LIN {X 0,Y 418.253,Z 298.382,A -85,B 0,C 180,E1 -10125.114,E2 -10125.114} C_VEL
LIN {X 0,Y 418.285,Z 298.384,A -85,B 0,C 180,E1 -10127.775,E2 -10127.775} C_VEL
LIN {X 0,Y 418.259,Z 298.386,A -85,B 0,C 180,E1 -10131.561,E2 -10131.561} C_VEL
LIN {X 0,Y 418.254,Z 298.387,A -85,B 0,C 180,E1 -10135.161,E2 -10135.161} C_VEL
LIN {X 0,Y 418.24,Z 298.388,A -85,B 0,C 180,E1 -10137.474,E2 -10137.474} C_VEL
LIN {X 0,Y 418.265,Z 298.384,A -85,B 0,C 180,E1 -10140.897,E2 -10140.897} C_VEL
LIN {X 0,Y 418.312,Z 298.534,A -85,B 0,C 180,E1 -10141.838,E2 -10141.838} C_VEL
LIN {X 0,Y 420.829,Z 310.049,A -85,B 0,C 180,E1 -10144.399,E2 -10144.399} C_VEL
LIN {X 0,Y 421.677,Z 315.896,A -85,B 0,C 180,E1 -10145.64,E2 -10145.64} C_VEL
LIN {X 0,Y 420.473,Z 332.793,A -85,B 0,C 180,E1 -10148.941,E2 -10148.941} C_VEL
LIN {X 0,Y 419.947,Z 341.283,A -85,B 0,C 180,E1 -10150.58,E2 -10150.58} C_VEL
LIN {X 0,Y 423.915,Z 364.649,A -85,B 0,C 180,E1 -10151.228,E2 -10151.228} C_VEL
LIN {X 0,Y 424.429,Z 370.899,A -85,B 0,C 180,E1 -10151.367,E2 -10151.367} C_VEL
LIN {X 0,Y 423.375,Z 450.721,A -85,B 0,C 180,E1 -10152.772,E2 -10152.772} C_VEL
LIN {X 0,Y 422.75,Z 464.397,A -85,B 0,C 180,E1 -10153.213,E2 -10153.213} C_VEL
LIN {X 0,Y 422.113,Z 476.708,A -85,B 0,C 180,E1 -10153.808,E2 -10153.808} C_VEL
LIN {X 0,Y 421.326,Z 487.75,A -85,B 0,C 180,E1 -10154.522,E2 -10154.522} C_VEL
LIN {X 0,Y 420.546,Z 499.288,A -85,B 0,C 180,E1 -10155.484,E2 -10155.484} C_VEL
LIN {X 0,Y 419.713,Z 509.697,A -85,B 0,C 180,E1 -10156.567,E2 -10156.567} C_VEL
LIN {X 0,Y 419.106,Z 518.223,A -85,B 0,C 180,E1 -10157.656,E2 -10157.656} C_VEL
LIN {X 0,Y 418.404,Z 526.105,A -85,B 0,C 180,E1 -10158.864,E2 -10158.864} C_VEL
LIN {X 0,Y 417.832,Z 533.825,A -85,B 0,C 180,E1 -10160.318,E2 -10160.318} C_VEL
LIN {X 0,Y 417.461,Z 540.039,A -85,B 0,C 180,E1 -10161.774,E2 -10161.774} C_VEL
LIN {X 0,Y 417.233,Z 544.991,A -85,B 0,C 180,E1 -10163.23,E2 -10163.23} C_VEL
LIN {X 0,Y 417.12,Z 548.824,A -85,B 0,C 180,E1 -10164.684,E2 -10164.684} C_VEL
LIN {X 0,Y 417.015,Z 551.638,A -85,B 0,C 180,E1 -10166.136,E2 -10166.136} C_VEL
LIN {X 0,Y 417.069,Z 553.918,A -85,B 0,C 180,E1 -10168.07,E2 -10168.07} C_VEL
LIN {X 0,Y 417.013,Z 554.462,A -85,B 0,C 180,E1 -10169.036,E2 -10169.036} C_VEL
LIN {X 0,Y 417.027,Z 554.574,A -85,B 0,C 180,E1 -10170.001,E2 -10170.001} C_VEL
LIN {X 0,Y 417.073,Z 553.627,A -85,B 0,C 180,E1 -10171.933,E2 -10171.933} C_VEL
LIN {X 0,Y 417.061,Z 552.561,A -85,B 0,C 180,E1 -10172.899,E2 -10172.899} C_VEL
LIN {X 0,Y 417.018,Z 551.035,A -85,B 0,C 180,E1 -10173.867,E2 -10173.867} C_VEL
LIN {X 0,Y 417.122,Z 547.958,A -85,B 0,C 180,E1 -10175.319,E2 -10175.319} C_VEL
LIN {X 0,Y 417.233,Z 543.806,A -85,B 0,C 180,E1 -10176.773,E2 -10176.773} C_VEL
LIN {X 0,Y 417.496,Z 537.449,A -85,B 0,C 180,E1 -10178.472,E2 -10178.472} C_VEL
LIN {X 0,Y 417.865,Z 530.518,A -85,B 0,C 180,E1 -10179.928,E2 -10179.928} C_VEL
LIN {X 0,Y 418.277,Z 523.434,A -85,B 0,C 180,E1 -10181.142,E2 -10181.142} C_VEL
LIN {X 0,Y 418.885,Z 514.891,A -85,B 0,C 180,E1 -10182.353,E2 -10182.353} C_VEL
LIN {X 0,Y 419.584,Z 504.318,A -85,B 0,C 180,E1 -10183.563,E2 -10183.563} C_VEL
LIN {X 0,Y 420.222,Z 492.389,A -85,B 0,C 180,E1 -10184.654,E2 -10184.654} C_VEL
LIN {X 0,Y 420.969,Z 480.36,A -85,B 0,C 180,E1 -10185.494,E2 -10185.494} C_VEL
LIN {X 0,Y 421.575,Z 467.817,A -85,B 0,C 180,E1 -10186.154,E2 -10186.154} C_VEL
LIN {X 0,Y 422.144,Z 454.764,A -85,B 0,C 180,E1 -10186.628,E2 -10186.628} C_VEL
LIN {X 0,Y 422.485,Z 438.987,A -85,B 0,C 180,E1 -10186.957,E2 -10186.957} C_VEL
LIN {X 0,Y 423.146,Z 367.635,A -85,B 0,C 180,E1 -10188.174,E2 -10188.174} C_VEL
LIN {X 0,Y 419.379,Z 341.81,A -85,B 0,C 180,E1 -10188.774,E2 -10188.774} C_VEL
LIN {X 0,Y 420.377,Z 324.387,A -85,B 0,C 180,E1 -10192.097,E2 -10192.097} C_VEL
LIN {X 0,Y 421.059,Z 313.774,A -85,B 0,C 180,E1 -10194.139,E2 -10194.139} C_VEL
LIN {X 0,Y 420.155,Z 307.557,A -85,B 0,C 180,E1 -10195.408,E2 -10195.408} C_VEL
LIN {X 0,Y 418.343,Z 298.376,A -85,B 0,C 180,E1 -10197.364,E2 -10197.364} C_VEL
LIN {X 0,Y 418.245,Z 298.384,A -85,B 0,C 180,E1 -10201.02,E2 -10201.02} C_VEL
LIN {X 0,Y 418.253,Z 298.382,A -85,B 0,C 180,E1 -10203.678,E2 -10203.678} C_VEL
LIN {X 0,Y 418.245,Z 298.382,A -85,B 0,C 180,E1 -10207.225,E2 -10207.225} C_VEL
LIN {X 0,Y 418.249,Z 298.382,A -85,B 0,C 180,E1 -10209.683,E2 -10209.683} C_VEL
LIN {X 0,Y 418.235,Z 298.388,A -85,B 0,C 180,E1 -10212.322,E2 -10212.322} C_VEL
LIN {X 0,Y 418.242,Z 298.384,A -85,B 0,C 180,E1 -10215.109,E2 -10215.109} C_VEL
LIN {X 0,Y 418.246,Z 298.382,A -85,B 0,C 180,E1 -10217.767,E2 -10217.767} C_VEL
LIN {X 0,Y 418.255,Z 298.386,A -85,B 0,C 180,E1 -10220.62,E2 -10220.62} C_VEL
LIN {X 0,Y 418.248,Z 298.381,A -85,B 0,C 180,E1 -10223.976,E2 -10223.976} C_VEL
LIN {X 0,Y 418.249,Z 298.384,A -85,B 0,C 180,E1 -10227.472,E2 -10227.472} C_VEL
LIN {X 0,Y 418.275,Z 298.383,A -85,B 0,C 180,E1 -10230.896,E2 -10230.896} C_VEL
LIN {X 0,Y 418.275,Z 298.378,A -85,B 0,C 180,E1 -10234.096,E2 -10234.096} C_VEL
LIN {X 0,Y 418.238,Z 298.389,A -85,B 0,C 180,E1 -10237.264,E2 -10237.264} C_VEL
LIN {X 0,Y 418.289,Z 298.376,A -85,B 0,C 180,E1 -10240.364,E2 -10240.364} C_VEL
LIN {X 0,Y 418.323,Z 298.378,A -85,B 0,C 180,E1 -10243.405,E2 -10243.405} C_VEL
LIN {X 0,Y 418.353,Z 298.369,A -85,B 0,C 180,E1 -10246.999,E2 -10246.999} C_VEL
LIN {X 0,Y 418.345,Z 298.371,A -85,B 0,C 180,E1 -10250.329,E2 -10250.329} C_VEL
LIN {X 0,Y 418.452,Z 298.357,A -85,B 0,C 180,E1 -10253.248,E2 -10253.248} C_VEL
LIN {X 0,Y 418.339,Z 298.37,A -85,B 0,C 180,E1 -10255.181,E2 -10255.181} C_VEL
LIN {X 0,Y 418.548,Z 298.352,A -85,B 0,C 180,E1 -10258.075,E2 -10258.075} C_VEL
LIN {X 0,Y 418.674,Z 298.335,A -85,B 0,C 180,E1 -10260,E2 -10260} C_VEL
LIN {X 0,Y 418.504,Z 298.35,A -85,B 0,C 180,E1 -10262.888,E2 -10262.888} C_VEL
LIN {X 0,Y 418.474,Z 298.355,A -85,B 0,C 180,E1 -10266.629,E2 -10266.629} C_VEL
LIN {X 0,Y 418.344,Z 298.37,A -85,B 0,C 180,E1 -10269.671,E2 -10269.671} C_VEL
LIN {X 0,Y 418.352,Z 298.371,A -85,B 0,C 180,E1 -10273,E2 -10273} C_VEL
LIN {X 0,Y 418.318,Z 298.38,A -85,B 0,C 180,E1 -10276.735,E2 -10276.735} C_VEL
LIN {X 0,Y 418.276,Z 298.378,A -85,B 0,C 180,E1 -10279.789,E2 -10279.789} C_VEL
LIN {X 0,Y 418.237,Z 298.389,A -85,B 0,C 180,E1 -10282.736,E2 -10282.736} C_VEL
LIN {X 0,Y 418.276,Z 298.378,A -85,B 0,C 180,E1 -10285.904,E2 -10285.904} C_VEL
LIN {X 0,Y 418.27,Z 298.385,A -85,B 0,C 180,E1 -10289.161,E2 -10289.161} C_VEL
LIN {X 0,Y 418.262,Z 298.383,A -85,B 0,C 180,E1 -10292.843,E2 -10292.843} C_VEL
LIN {X 0,Y 418.248,Z 298.381,A -85,B 0,C 180,E1 -10296.237,E2 -10296.237} C_VEL
LIN {X 0,Y 418.255,Z 298.385,A -85,B 0,C 180,E1 -10299.681,E2 -10299.681} C_VEL
LIN {X 0,Y 418.234,Z 298.383,A -85,B 0,C 180,E1 -10302.32,E2 -10302.32} C_VEL
LIN {X 0,Y 418.24,Z 298.385,A -85,B 0,C 180,E1 -10305.108,E2 -10305.108} C_VEL
LIN {X 0,Y 418.243,Z 298.389,A -85,B 0,C 180,E1 -10307.766,E2 -10307.766} C_VEL
LIN {X 0,Y 418.249,Z 298.381,A -85,B 0,C 180,E1 -10310.62,E2 -10310.62} C_VEL
LIN {X 0,Y 418.247,Z 298.388,A -85,B 0,C 180,E1 -10313.975,E2 -10313.975} C_VEL
LIN {X 0,Y 418.261,Z 298.38,A -85,B 0,C 180,E1 -10317.155,E2 -10317.155} C_VEL
LIN {X 0,Y 418.272,Z 298.379,A -85,B 0,C 180,E1 -10320.894,E2 -10320.894} C_VEL
LIN {X 0,Y 418.272,Z 298.385,A -85,B 0,C 180,E1 -10324.095,E2 -10324.095} C_VEL
LIN {X 0,Y 418.241,Z 298.382,A -85,B 0,C 180,E1 -10327.263,E2 -10327.263} C_VEL
LIN {X 0,Y 418.319,Z 298.38,A -85,B 0,C 180,E1 -10330.365,E2 -10330.365} C_VEL
LIN {X 0,Y 418.32,Z 298.372,A -85,B 0,C 180,E1 -10333.403,E2 -10333.403} C_VEL
LIN {X 0,Y 418.348,Z 298.372,A -85,B 0,C 180,E1 -10336.998,E2 -10336.998} C_VEL
LIN {X 0,Y 418.34,Z 298.373,A -85,B 0,C 180,E1 -10340.327,E2 -10340.327} C_VEL
LIN {X 0,Y 418.457,Z 298.388,A -85,B 0,C 180,E1 -10343.121,E2 -10343.121} C_VEL
LIN {X 0,Y 419.862,Z 307.44,A -85,B 0,C 180,E1 -10345.198,E2 -10345.198} C_VEL
LIN {X 0,Y 419.717,Z 312.544,A -85,B 0,C 180,E1 -10346.308,E2 -10346.308} C_VEL
LIN {X 0,Y 423.532,Z 333.046,A -85,B 0,C 180,E1 -10346.824,E2 -10346.824} C_VEL
LIN {X 0,Y 422.396,Z 420.515,A -85,B 0,C 180,E1 -10348.335,E2 -10348.335} C_VEL
LIN {X 0,Y 422.141,Z 430.007,A -85,B 0,C 180,E1 -10348.618,E2 -10348.618} C_VEL
LIN {X 0,Y 421.418,Z 435.689,A -85,B 0,C 180,E1 -10348.815,E2 -10348.815} C_VEL
LIN {X 0,Y 418.342,Z 444.777,A -85,B 0,C 180,E1 -10349.157,E2 -10349.157} C_VEL
LIN {X 0,Y 415.083,Z 453.573,A -85,B 0,C 180,E1 -10349.603,E2 -10349.603} C_VEL
LIN {X 0,Y 414.083,Z 458.797,A -85,B 0,C 180,E1 -10349.96,E2 -10349.96} C_VEL
LIN {X 0,Y 413.337,Z 470.545,A -85,B 0,C 180,E1 -10350.973,E2 -10350.973} C_VEL
LIN {X 0,Y 412.59,Z 480.693,A -85,B 0,C 180,E1 -10352.073,E2 -10352.073} C_VEL
LIN {X 0,Y 411.883,Z 490.629,A -85,B 0,C 180,E1 -10353.422,E2 -10353.422} C_VEL
LIN {X 0,Y 411.278,Z 499.38,A -85,B 0,C 180,E1 -10354.9,E2 -10354.9} C_VEL
LIN {X 0,Y 410.901,Z 506.355,A -85,B 0,C 180,E1 -10356.382,E2 -10356.382} C_VEL
LIN {X 0,Y 410.522,Z 511.96,A -85,B 0,C 180,E1 -10357.87,E2 -10357.87} C_VEL
LIN {X 0,Y 410.249,Z 516.367,A -85,B 0,C 180,E1 -10359.365,E2 -10359.365} C_VEL
LIN {X 0,Y 410.086,Z 519.69,A -85,B 0,C 180,E1 -10360.865,E2 -10360.865} C_VEL
LIN {X 0,Y 409.94,Z 521.881,A -85,B 0,C 180,E1 -10362.258,E2 -10362.258} C_VEL
LIN {X 0,Y 409.84,Z 523.379,A -85,B 0,C 180,E1 -10363.889,E2 -10363.889} C_VEL
LIN {X 0,Y 409.853,Z 523.751,A -85,B 0,C 180,E1 -10364.903,E2 -10364.903} C_VEL
LIN {X 0,Y 409.855,Z 523.645,A -85,B 0,C 180,E1 -10366.207,E2 -10366.207} C_VEL
LIN {X 0,Y 409.93,Z 522.359,A -85,B 0,C 180,E1 -10367.973,E2 -10367.973} C_VEL
LIN {X 0,Y 410.158,Z 520.14,A -85,B 0,C 180,E1 -10369.539,E2 -10369.539} C_VEL
LIN {X 0,Y 410.355,Z 516.918,A -85,B 0,C 180,E1 -10371.077,E2 -10371.077} C_VEL
LIN {X 0,Y 410.73,Z 512.238,A -85,B 0,C 180,E1 -10372.716,E2 -10372.716} C_VEL
LIN {X 0,Y 411.197,Z 506.699,A -85,B 0,C 180,E1 -10374.215,E2 -10374.215} C_VEL
LIN {X 0,Y 411.84,Z 499.345,A -85,B 0,C 180,E1 -10375.793,E2 -10375.793} C_VEL
LIN {X 0,Y 412.55,Z 491.704,A -85,B 0,C 180,E1 -10377.108,E2 -10377.108} C_VEL
LIN {X 0,Y 413.388,Z 482.313,A -85,B 0,C 180,E1 -10378.424,E2 -10378.424} C_VEL
LIN {X 0,Y 414.076,Z 473.077,A -85,B 0,C 180,E1 -10379.484,E2 -10379.484} C_VEL
LIN {X 0,Y 414.997,Z 461.664,A -85,B 0,C 180,E1 -10380.532,E2 -10380.532} C_VEL
LIN {X 0,Y 415.769,Z 449.638,A -85,B 0,C 180,E1 -10381.387,E2 -10381.387} C_VEL
LIN {X 0,Y 416.379,Z 437.805,A -85,B 0,C 180,E1 -10382.022,E2 -10382.022} C_VEL
LIN {X 0,Y 416.819,Z 425.374,A -85,B 0,C 180,E1 -10382.496,E2 -10382.496} C_VEL
LIN {X 0,Y 417.163,Z 410.81,A -85,B 0,C 180,E1 -10382.818,E2 -10382.818} C_VEL
LIN {X 0,Y 418.122,Z 333.025,A -85,B 0,C 180,E1 -10384.188,E2 -10384.188} C_VEL
LIN {X 0,Y 414.056,Z 315.081,A -85,B 0,C 180,E1 -10384.753,E2 -10384.753} C_VEL
LIN {X 0,Y 413.542,Z 312.748,A -85,B 0,C 180,E1 -10384.864,E2 -10384.864} C_VEL
LIN {X 0,Y 413.307,Z 309.399,A -85,B 0,C 180,E1 -10385.616,E2 -10385.616} C_VEL
LIN {X 0,Y 411.168,Z 299.271,A -85,B 0,C 180,E1 -10388.079,E2 -10388.079} C_VEL
LIN {X 0,Y 411.136,Z 299.271,A -85,B 0,C 180,E1 -10391.224,E2 -10391.224} C_VEL
LIN {X 0,Y 411.163,Z 299.268,A -85,B 0,C 180,E1 -10394.489,E2 -10394.489} C_VEL
LIN {X 0,Y 411.151,Z 299.269,A -85,B 0,C 180,E1 -10398.192,E2 -10398.192} C_VEL
LIN {X 0,Y 411.178,Z 299.27,A -85,B 0,C 180,E1 -10401.833,E2 -10401.833} C_VEL
LIN {X 0,Y 411.195,Z 299.251,A -85,B 0,C 180,E1 -10405.121,E2 -10405.121} C_VEL
LIN {X 0,Y 411.152,Z 299.268,A -85,B 0,C 180,E1 -10408.002,E2 -10408.002} C_VEL
LIN {X 0,Y 411.181,Z 299.266,A -85,B 0,C 180,E1 -10411.407,E2 -10411.407} C_VEL
LIN {X 0,Y 411.213,Z 299.256,A -85,B 0,C 180,E1 -10414.929,E2 -10414.929} C_VEL
LIN {X 0,Y 411.19,Z 299.266,A -85,B 0,C 180,E1 -10417.913,E2 -10417.913} C_VEL
LIN {X 0,Y 411.207,Z 299.26,A -85,B 0,C 180,E1 -10421.051,E2 -10421.051} C_VEL
LIN {X 0,Y 411.239,Z 299.256,A -85,B 0,C 180,E1 -10424.131,E2 -10424.131} C_VEL
LIN {X 0,Y 411.288,Z 299.246,A -85,B 0,C 180,E1 -10427.165,E2 -10427.165} C_VEL
LIN {X 0,Y 411.289,Z 299.254,A -85,B 0,C 180,E1 -10430.161,E2 -10430.161} C_VEL
LIN {X 0,Y 411.408,Z 299.228,A -85,B 0,C 180,E1 -10433.132,E2 -10433.132} C_VEL
LIN {X 0,Y 411.291,Z 299.25,A -85,B 0,C 180,E1 -10435.099,E2 -10435.099} C_VEL
LIN {X 0,Y 411.497,Z 299.22,A -85,B 0,C 180,E1 -10438.043,E2 -10438.043} C_VEL
LIN {X 0,Y 411.626,Z 299.206,A -85,B 0,C 180,E1 -10440,E2 -10440} C_VEL
LIN {X 0,Y 411.443,Z 299.224,A -85,B 0,C 180,E1 -10442.938,E2 -10442.938} C_VEL
LIN {X 0,Y 411.444,Z 299.23,A -85,B 0,C 180,E1 -10446.867,E2 -10446.867} C_VEL
LIN {X 0,Y 411.341,Z 299.24,A -85,B 0,C 180,E1 -10448.846,E2 -10448.846} C_VEL
LIN {X 0,Y 411.271,Z 299.251,A -85,B 0,C 180,E1 -10451.833,E2 -10451.833} C_VEL
LIN {X 0,Y 411.246,Z 299.254,A -85,B 0,C 180,E1 -10454.853,E2 -10454.853} C_VEL
LIN {X 0,Y 411.239,Z 299.252,A -85,B 0,C 180,E1 -10457.916,E2 -10457.916} C_VEL
LIN {X 0,Y 411.183,Z 299.269,A -85,B 0,C 180,E1 -10461.035,E2 -10461.035} C_VEL
LIN {X 0,Y 411.214,Z 299.254,A -85,B 0,C 180,E1 -10464.216,E2 -10464.216} C_VEL
LIN {X 0,Y 411.248,Z 299.252,A -85,B 0,C 180,E1 -10467.479,E2 -10467.479} C_VEL
LIN {X 0,Y 411.191,Z 299.266,A -85,B 0,C 180,E1 -10470.848,E2 -10470.848} C_VEL
LIN {X 0,Y 411.196,Z 299.263,A -85,B 0,C 180,E1 -10474.335,E2 -10474.335} C_VEL
LIN {X 0,Y 411.195,Z 299.264,A -85,B 0,C 180,E1 -10477.974,E2 -10477.974} C_VEL
LIN {X 0,Y 411.192,Z 299.269,A -85,B 0,C 180,E1 -10481.236,E2 -10481.236} C_VEL
LIN {X 0,Y 411.18,Z 299.262,A -85,B 0,C 180,E1 -10484.49,E2 -10484.49} C_VEL
LIN {X 0,Y 411.222,Z 299.257,A -85,B 0,C 180,E1 -10487.299,E2 -10487.299} C_VEL
LIN {X 0,Y 411.224,Z 299.257,A -85,B 0,C 180,E1 -10490.779,E2 -10490.779} C_VEL
LIN {X 0,Y 411.194,Z 299.266,A -85,B 0,C 180,E1 -10494.473,E2 -10494.473} C_VEL
LIN {X 0,Y 411.202,Z 299.262,A -85,B 0,C 180,E1 -10496.875,E2 -10496.875} C_VEL
LIN {X 0,Y 411.229,Z 299.259,A -85,B 0,C 180,E1 -10500.646,E2 -10500.646} C_VEL
LIN {X 0,Y 411.294,Z 299.423,A -85,B 0,C 180,E1 -10501.494,E2 -10501.494} C_VEL
LIN {X 0,Y 413.863,Z 311.135,A -85,B 0,C 180,E1 -10504.161,E2 -10504.161} C_VEL
LIN {X 0,Y 414.801,Z 317.201,A -85,B 0,C 180,E1 -10505.476,E2 -10505.476} C_VEL
LIN {X 0,Y 413.55,Z 334.086,A -85,B 0,C 180,E1 -10508.832,E2 -10508.832} C_VEL
LIN {X 0,Y 413.076,Z 341.056,A -85,B 0,C 180,E1 -10510.203,E2 -10510.203} C_VEL
LIN {X 0,Y 417.161,Z 364.626,A -85,B 0,C 180,E1 -10510.867,E2 -10510.867} C_VEL
LIN {X 0,Y 417.815,Z 370.654,A -85,B 0,C 180,E1 -10511.013,E2 -10511.013} C_VEL
LIN {X 0,Y 416.687,Z 449.899,A -85,B 0,C 180,E1 -10512.423,E2 -10512.423} C_VEL
LIN {X 0,Y 416.097,Z 463.747,A -85,B 0,C 180,E1 -10512.873,E2 -10512.873} C_VEL
LIN {X 0,Y 415.395,Z 476.174,A -85,B 0,C 180,E1 -10513.476,E2 -10513.476} C_VEL
LIN {X 0,Y 414.513,Z 488.07,A -85,B 0,C 180,E1 -10514.261,E2 -10514.261} C_VEL
LIN {X 0,Y 413.672,Z 499.486,A -85,B 0,C 180,E1 -10515.238,E2 -10515.238} C_VEL
LIN {X 0,Y 412.786,Z 509.803,A -85,B 0,C 180,E1 -10516.337,E2 -10516.337} C_VEL
LIN {X 0,Y 412.147,Z 518.256,A -85,B 0,C 180,E1 -10517.444,E2 -10517.444} C_VEL
LIN {X 0,Y 411.295,Z 527.442,A -85,B 0,C 180,E1 -10518.918,E2 -10518.918} C_VEL
LIN {X 0,Y 410.739,Z 534.855,A -85,B 0,C 180,E1 -10520.398,E2 -10520.398} C_VEL
LIN {X 0,Y 410.321,Z 541.71,A -85,B 0,C 180,E1 -10522.126,E2 -10522.126} C_VEL
LIN {X 0,Y 410.042,Z 546.679,A -85,B 0,C 180,E1 -10523.777,E2 -10523.777} C_VEL
LIN {X 0,Y 410.018,Z 549.704,A -85,B 0,C 180,E1 -10525.085,E2 -10525.085} C_VEL
LIN {X 0,Y 409.928,Z 552.753,A -85,B 0,C 180,E1 -10527.053,E2 -10527.053} C_VEL
LIN {X 0,Y 409.996,Z 553.685,A -85,B 0,C 180,E1 -10528.037,E2 -10528.037} C_VEL
LIN {X 0,Y 409.938,Z 554.208,A -85,B 0,C 180,E1 -10529.019,E2 -10529.019} C_VEL
LIN {X 0,Y 409.948,Z 554.302,A -85,B 0,C 180,E1 -10530.001,E2 -10530.001} C_VEL
LIN {X 0,Y 410.001,Z 553.331,A -85,B 0,C 180,E1 -10531.966,E2 -10531.966} C_VEL
LIN {X 0,Y 409.959,Z 552.242,A -85,B 0,C 180,E1 -10532.949,E2 -10532.949} C_VEL
LIN {X 0,Y 409.937,Z 550.698,A -85,B 0,C 180,E1 -10533.934,E2 -10533.934} C_VEL
LIN {X 0,Y 410.019,Z 547.59,A -85,B 0,C 180,E1 -10535.411,E2 -10535.411} C_VEL
LIN {X 0,Y 410.165,Z 543.409,A -85,B 0,C 180,E1 -10536.89,E2 -10536.89} C_VEL
LIN {X 0,Y 410.426,Z 537.017,A -85,B 0,C 180,E1 -10538.619,E2 -10538.619} C_VEL
LIN {X 0,Y 410.806,Z 530.047,A -85,B 0,C 180,E1 -10540.101,E2 -10540.101} C_VEL
LIN {X 0,Y 411.379,Z 521.302,A -85,B 0,C 180,E1 -10541.581,E2 -10541.581} C_VEL
LIN {X 0,Y 412.001,Z 512.334,A -85,B 0,C 180,E1 -10542.814,E2 -10542.814} C_VEL
LIN {X 0,Y 412.653,Z 502.834,A -85,B 0,C 180,E1 -10543.883,E2 -10543.883} C_VEL
LIN {X 0,Y 413.329,Z 491.621,A -85,B 0,C 180,E1 -10544.904,E2 -10544.904} C_VEL
LIN {X 0,Y 414.103,Z 479.435,A -85,B 0,C 180,E1 -10545.758,E2 -10545.758} C_VEL
LIN {X 0,Y 414.764,Z 466.689,A -85,B 0,C 180,E1 -10546.426,E2 -10546.426} C_VEL
LIN {X 0,Y 415.272,Z 454.102,A -85,B 0,C 180,E1 -10546.88,E2 -10546.88} C_VEL
LIN {X 0,Y 415.595,Z 438.077,A -85,B 0,C 180,E1 -10547.215,E2 -10547.215} C_VEL
LIN {X 0,Y 416.208,Z 367.341,A -85,B 0,C 180,E1 -10548.443,E2 -10548.443} C_VEL
LIN {X 0,Y 412.425,Z 341.549,A -85,B 0,C 180,E1 -10549.054,E2 -10549.054} C_VEL
LIN {X 0,Y 413.409,Z 325.2,A -85,B 0,C 180,E1 -10552.227,E2 -10552.227} C_VEL
LIN {X 0,Y 414.081,Z 314.581,A -85,B 0,C 180,E1 -10554.306,E2 -10554.306} C_VEL
LIN {X 0,Y 412.855,Z 307.049,A -85,B 0,C 180,E1 -10555.878,E2 -10555.878} C_VEL
LIN {X 0,Y 411.318,Z 299.252,A -85,B 0,C 180,E1 -10557.578,E2 -10557.578} C_VEL
LIN {X 0,Y 411.188,Z 299.262,A -85,B 0,C 180,E1 -10561.284,E2 -10561.284} C_VEL
LIN {X 0,Y 411.211,Z 299.265,A -85,B 0,C 180,E1 -10564.334,E2 -10564.334} C_VEL
LIN {X 0,Y 411.196,Z 299.263,A -85,B 0,C 180,E1 -10567.975,E2 -10567.975} C_VEL
LIN {X 0,Y 411.169,Z 299.264,A -85,B 0,C 180,E1 -10571.229,E2 -10571.229} C_VEL
LIN {X 0,Y 411.182,Z 299.268,A -85,B 0,C 180,E1 -10574.491,E2 -10574.491} C_VEL
LIN {X 0,Y 411.183,Z 299.263,A -85,B 0,C 180,E1 -10578.195,E2 -10578.195} C_VEL
LIN {X 0,Y 411.22,Z 299.264,A -85,B 0,C 180,E1 -10580.776,E2 -10580.776} C_VEL
LIN {X 0,Y 411.201,Z 299.262,A -85,B 0,C 180,E1 -10584.471,E2 -10584.471} C_VEL
LIN {X 0,Y 411.211,Z 299.264,A -85,B 0,C 180,E1 -10586.874,E2 -10586.874} C_VEL
LIN {X 0,Y 411.239,Z 299.256,A -85,B 0,C 180,E1 -10590.644,E2 -10590.644} C_VEL
LIN {X 0,Y 411.244,Z 299.257,A -85,B 0,C 180,E1 -10593.619,E2 -10593.619} C_VEL
LIN {X 0,Y 411.203,Z 299.261,A -85,B 0,C 180,E1 -10596.852,E2 -10596.852} C_VEL
LIN {X 0,Y 411.221,Z 299.258,A -85,B 0,C 180,E1 -10600.051,E2 -10600.051} C_VEL
LIN {X 0,Y 411.27,Z 299.253,A -85,B 0,C 180,E1 -10603.131,E2 -10603.131} C_VEL
LIN {X 0,Y 411.312,Z 299.246,A -85,B 0,C 180,E1 -10606.896,E2 -10606.896} C_VEL
LIN {X 0,Y 411.297,Z 299.25,A -85,B 0,C 180,E1 -10610.161,E2 -10610.161} C_VEL
LIN {X 0,Y 411.401,Z 299.235,A -85,B 0,C 180,E1 -10613.132,E2 -10613.132} C_VEL
LIN {X 0,Y 411.309,Z 299.246,A -85,B 0,C 180,E1 -10615.099,E2 -10615.099} C_VEL
LIN {X 0,Y 411.517,Z 299.228,A -85,B 0,C 180,E1 -10618.042,E2 -10618.042} C_VEL
LIN {X 0,Y 411.643,Z 299.211,A -85,B 0,C 180,E1 -10620,E2 -10620} C_VEL
LIN {X 0,Y 411.461,Z 299.227,A -85,B 0,C 180,E1 -10622.937,E2 -10622.937} C_VEL
LIN {X 0,Y 411.437,Z 299.23,A -85,B 0,C 180,E1 -10626.629,E2 -10626.629} C_VEL
LIN {X 0,Y 411.324,Z 299.246,A -85,B 0,C 180,E1 -10628.846,E2 -10628.846} C_VEL
LIN {X 0,Y 411.288,Z 299.249,A -85,B 0,C 180,E1 -10631.832,E2 -10631.832} C_VEL
LIN {X 0,Y 411.266,Z 299.256,A -85,B 0,C 180,E1 -10634.852,E2 -10634.852} C_VEL
LIN {X 0,Y 411.251,Z 299.253,A -85,B 0,C 180,E1 -10637.915,E2 -10637.915} C_VEL
LIN {X 0,Y 411.201,Z 299.264,A -85,B 0,C 180,E1 -10641.034,E2 -10641.034} C_VEL
LIN {X 0,Y 411.226,Z 299.257,A -85,B 0,C 180,E1 -10644.215,E2 -10644.215} C_VEL
LIN {X 0,Y 411.264,Z 299.254,A -85,B 0,C 180,E1 -10647.477,E2 -10647.477} C_VEL
LIN {X 0,Y 411.194,Z 299.264,A -85,B 0,C 180,E1 -10650.847,E2 -10650.847} C_VEL
LIN {X 0,Y 411.21,Z 299.258,A -85,B 0,C 180,E1 -10654.333,E2 -10654.333} C_VEL
LIN {X 0,Y 411.199,Z 299.261,A -85,B 0,C 180,E1 -10657.973,E2 -10657.973} C_VEL
LIN {X 0,Y 411.186,Z 299.261,A -85,B 0,C 180,E1 -10660.503,E2 -10660.503} C_VEL
LIN {X 0,Y 411.178,Z 299.265,A -85,B 0,C 180,E1 -10663.133,E2 -10663.133} C_VEL
LIN {X 0,Y 411.172,Z 299.267,A -85,B 0,C 180,E1 -10665.88,E2 -10665.88} C_VEL
LIN {X 0,Y 411.167,Z 299.263,A -85,B 0,C 180,E1 -10668.771,E2 -10668.771} C_VEL
LIN {X 0,Y 411.195,Z 299.265,A -85,B 0,C 180,E1 -10672.025,E2 -10672.025} C_VEL
LIN {X 0,Y 411.21,Z 299.263,A -85,B 0,C 180,E1 -10675.666,E2 -10675.666} C_VEL
LIN {X 0,Y 411.193,Z 299.26,A -85,B 0,C 180,E1 -10679.151,E2 -10679.151} C_VEL
LIN {X 0,Y 411.262,Z 299.255,A -85,B 0,C 180,E1 -10682.521,E2 -10682.521} C_VEL
LIN {X 0,Y 411.229,Z 299.258,A -85,B 0,C 180,E1 -10685.783,E2 -10685.783} C_VEL
LIN {X 0,Y 411.205,Z 299.26,A -85,B 0,C 180,E1 -10688.965,E2 -10688.965} C_VEL
LIN {X 0,Y 411.255,Z 299.255,A -85,B 0,C 180,E1 -10692.084,E2 -10692.084} C_VEL
LIN {X 0,Y 411.262,Z 299.253,A -85,B 0,C 180,E1 -10695.146,E2 -10695.146} C_VEL
LIN {X 0,Y 411.286,Z 299.251,A -85,B 0,C 180,E1 -10698.166,E2 -10698.166} C_VEL
LIN {X 0,Y 411.438,Z 299.236,A -85,B 0,C 180,E1 -10702.191,E2 -10702.191} C_VEL
LIN {X 0,Y 411.4,Z 299.304,A -85,B 0,C 180,E1 -10702.941,E2 -10702.941} C_VEL
LIN {X 0,Y 412.773,Z 307.583,A -85,B 0,C 180,E1 -10704.87,E2 -10704.87} C_VEL
LIN {X 0,Y 412.749,Z 312.82,A -85,B 0,C 180,E1 -10706.032,E2 -10706.032} C_VEL
LIN {X 0,Y 416.688,Z 333.567,A -85,B 0,C 180,E1 -10706.566,E2 -10706.566} C_VEL
LIN {X 0,Y 415.539,Z 420.703,A -85,B 0,C 180,E1 -10708.094,E2 -10708.094} C_VEL
LIN {X 0,Y 415.127,Z 434.046,A -85,B 0,C 180,E1 -10708.532,E2 -10708.532} C_VEL
LIN {X 0,Y 414.743,Z 446.232,A -85,B 0,C 180,E1 -10709.126,E2 -10709.126} C_VEL
LIN {X 0,Y 414.174,Z 457.555,A -85,B 0,C 180,E1 -10709.865,E2 -10709.865} C_VEL
LIN {X 0,Y 414.083,Z 458.797,A -85,B 0,C 180,E1 -10709.96,E2 -10709.96} C_VEL
LIN {X 0,Y 413.066,Z 463.961,A -85,B 0,C 180,E1 -10710.35,E2 -10710.35} C_VEL
LIN {X 0,Y 409.673,Z 472.006,A -85,B 0,C 180,E1 -10711.003,E2 -10711.003} C_VEL
LIN {X 0,Y 406.329,Z 479.625,A -85,B 0,C 180,E1 -10711.754,E2 -10711.754} C_VEL
LIN {X 0,Y 405.392,Z 484.022,A -85,B 0,C 180,E1 -10712.289,E2 -10712.289} C_VEL
LIN {X 0,Y 404.774,Z 492.295,A -85,B 0,C 180,E1 -10713.482,E2 -10713.482} C_VEL
LIN {X 0,Y 404.167,Z 500.728,A -85,B 0,C 180,E1 -10714.986,E2 -10714.986} C_VEL
LIN {X 0,Y 403.806,Z 507.496,A -85,B 0,C 180,E1 -10716.494,E2 -10716.494} C_VEL
LIN {X 0,Y 403.404,Z 512.934,A -85,B 0,C 180,E1 -10718.01,E2 -10718.01} C_VEL
LIN {X 0,Y 403.138,Z 517.182,A -85,B 0,C 180,E1 -10719.531,E2 -10719.531} C_VEL
LIN {X 0,Y 402.991,Z 520.352,A -85,B 0,C 180,E1 -10721.058,E2 -10721.058} C_VEL
LIN {X 0,Y 402.86,Z 522.234,A -85,B 0,C 180,E1 -10722.331,E2 -10722.331} C_VEL
LIN {X 0,Y 402.763,Z 523.753,A -85,B 0,C 180,E1 -10724.138,E2 -10724.138} C_VEL
LIN {X 0,Y 402.764,Z 524.055,A -85,B 0,C 180,E1 -10725.172,E2 -10725.172} C_VEL
LIN {X 0,Y 402.761,Z 523.891,A -85,B 0,C 180,E1 -10726.317,E2 -10726.317} C_VEL
LIN {X 0,Y 402.868,Z 522.373,A -85,B 0,C 180,E1 -10728.299,E2 -10728.299} C_VEL
LIN {X 0,Y 403.089,Z 520.356,A -85,B 0,C 180,E1 -10729.694,E2 -10729.694} C_VEL
LIN {X 0,Y 403.35,Z 516.623,A -85,B 0,C 180,E1 -10731.461,E2 -10731.461} C_VEL
LIN {X 0,Y 403.749,Z 511.96,A -85,B 0,C 180,E1 -10733.071,E2 -10733.071} C_VEL
LIN {X 0,Y 404.321,Z 506.024,A -85,B 0,C 180,E1 -10734.654,E2 -10734.654} C_VEL
LIN {X 0,Y 405.024,Z 498.369,A -85,B 0,C 180,E1 -10736.26,E2 -10736.26} C_VEL
LIN {X 0,Y 405.791,Z 490.47,A -85,B 0,C 180,E1 -10737.598,E2 -10737.598} C_VEL
LIN {X 0,Y 406.719,Z 480.765,A -85,B 0,C 180,E1 -10738.934,E2 -10738.934} C_VEL
LIN {X 0,Y 407.505,Z 471.104,A -85,B 0,C 180,E1 -10740.008,E2 -10740.008} C_VEL
LIN {X 0,Y 408.482,Z 459.012,A -85,B 0,C 180,E1 -10741.073,E2 -10741.073} C_VEL
LIN {X 0,Y 409.208,Z 447.266,A -85,B 0,C 180,E1 -10741.876,E2 -10741.876} C_VEL
LIN {X 0,Y 409.873,Z 434.799,A -85,B 0,C 180,E1 -10742.499,E2 -10742.499} C_VEL
LIN {X 0,Y 410.3,Z 421.299,A -85,B 0,C 180,E1 -10742.957,E2 -10742.957} C_VEL
LIN {X 0,Y 411.592,Z 334.29,A -85,B 0,C 180,E1 -10744.539,E2 -10744.539} C_VEL
LIN {X 0,Y 407.491,Z 316.233,A -85,B 0,C 180,E1 -10745.124,E2 -10745.124} C_VEL
LIN {X 0,Y 406.661,Z 313.063,A -85,B 0,C 180,E1 -10745.261,E2 -10745.261} C_VEL
LIN {X 0,Y 404.974,Z 304.151,A -85,B 0,C 180,E1 -10747.399,E2 -10747.399} C_VEL
LIN {X 0,Y 404.134,Z 300.146,A -85,B 0,C 180,E1 -10748.417,E2 -10748.417} C_VEL
LIN {X 0,Y 404.094,Z 300.15,A -85,B 0,C 180,E1 -10751.595,E2 -10751.595} C_VEL
LIN {X 0,Y 404.132,Z 300.144,A -85,B 0,C 180,E1 -10754.52,E2 -10754.52} C_VEL
LIN {X 0,Y 404.112,Z 300.145,A -85,B 0,C 180,E1 -10757.293,E2 -10757.293} C_VEL
LIN {X 0,Y 404.12,Z 300.147,A -85,B 0,C 180,E1 -10759.95,E2 -10759.95} C_VEL
LIN {X 0,Y 404.119,Z 300.146,A -85,B 0,C 180,E1 -10763.125,E2 -10763.125} C_VEL
LIN {X 0,Y 404.131,Z 300.145,A -85,B 0,C 180,E1 -10766.187,E2 -10766.187} C_VEL
LIN {X 0,Y 404.131,Z 300.146,A -85,B 0,C 180,E1 -10769.714,E2 -10769.714} C_VEL
LIN {X 0,Y 404.12,Z 300.143,A -85,B 0,C 180,E1 -10773.118,E2 -10773.118} C_VEL
LIN {X 0,Y 404.143,Z 300.142,A -85,B 0,C 180,E1 -10776.424,E2 -10776.424} C_VEL
LIN {X 0,Y 404.177,Z 300.135,A -85,B 0,C 180,E1 -10779.874,E2 -10779.874} C_VEL
LIN {X 0,Y 404.201,Z 300.127,A -85,B 0,C 180,E1 -10782.993,E2 -10782.993} C_VEL
LIN {X 0,Y 404.268,Z 300.121,A -85,B 0,C 180,E1 -10786.939,E2 -10786.939} C_VEL
LIN {X 0,Y 404.251,Z 300.128,A -85,B 0,C 180,E1 -10789.988,E2 -10789.988} C_VEL
LIN {X 0,Y 404.354,Z 300.107,A -85,B 0,C 180,E1 -10793.012,E2 -10793.012} C_VEL
LIN {X 0,Y 404.261,Z 300.126,A -85,B 0,C 180,E1 -10795.014,E2 -10795.014} C_VEL
LIN {X 0,Y 404.466,Z 300.096,A -85,B 0,C 180,E1 -10798.009,E2 -10798.009} C_VEL
LIN {X 0,Y 404.596,Z 300.082,A -85,B 0,C 180,E1 -10800,E2 -10800} C_VEL
LIN {X 0,Y 404.402,Z 300.1,A -85,B 0,C 180,E1 -10802.989,E2 -10802.989} C_VEL
LIN {X 0,Y 404.396,Z 300.107,A -85,B 0,C 180,E1 -10806.988,E2 -10806.988} C_VEL
LIN {X 0,Y 404.246,Z 300.124,A -85,B 0,C 180,E1 -10810.012,E2 -10810.012} C_VEL
LIN {X 0,Y 404.253,Z 300.119,A -85,B 0,C 180,E1 -10813.212,E2 -10813.212} C_VEL
LIN {X 0,Y 404.202,Z 300.135,A -85,B 0,C 180,E1 -10817.008,E2 -10817.008} C_VEL
LIN {X 0,Y 404.151,Z 300.138,A -85,B 0,C 180,E1 -10820.353,E2 -10820.353} C_VEL
LIN {X 0,Y 404.157,Z 300.134,A -85,B 0,C 180,E1 -10823.576,E2 -10823.576} C_VEL
LIN {X 0,Y 404.172,Z 300.138,A -85,B 0,C 180,E1 -10825.767,E2 -10825.767} C_VEL
LIN {X 0,Y 404.186,Z 300.128,A -85,B 0,C 180,E1 -10828.001,E2 -10828.001} C_VEL
LIN {X 0,Y 404.137,Z 300.139,A -85,B 0,C 180,E1 -10831.561,E2 -10831.561} C_VEL
LIN {X 0,Y 404.175,Z 300.142,A -85,B 0,C 180,E1 -10835.017,E2 -10835.017} C_VEL
LIN {X 0,Y 404.154,Z 300.141,A -85,B 0,C 180,E1 -10838.757,E2 -10838.757} C_VEL
LIN {X 0,Y 404.142,Z 300.144,A -85,B 0,C 180,E1 -10841.606,E2 -10841.606} C_VEL
LIN {X 0,Y 404.149,Z 300.138,A -85,B 0,C 180,E1 -10844.525,E2 -10844.525} C_VEL
LIN {X 0,Y 404.2,Z 300.132,A -85,B 0,C 180,E1 -10847.307,E2 -10847.307} C_VEL
LIN {X 0,Y 404.162,Z 300.134,A -85,B 0,C 180,E1 -10849.957,E2 -10849.957} C_VEL
LIN {X 0,Y 404.135,Z 300.143,A -85,B 0,C 180,E1 -10853.126,E2 -10853.126} C_VEL
LIN {X 0,Y 404.14,Z 300.14,A -85,B 0,C 180,E1 -10856.19,E2 -10856.19} C_VEL
LIN {X 0,Y 404.141,Z 300.147,A -85,B 0,C 180,E1 -10859.717,E2 -10859.717} C_VEL
LIN {X 0,Y 404.229,Z 300.26,A -85,B 0,C 180,E1 -10861.12,E2 -10861.12} C_VEL
LIN {X 0,Y 406.906,Z 312.248,A -85,B 0,C 180,E1 -10863.914,E2 -10863.914} C_VEL
LIN {X 0,Y 407.914,Z 318.512,A -85,B 0,C 180,E1 -10865.306,E2 -10865.306} C_VEL
LIN {X 0,Y 406.629,Z 335.39,A -85,B 0,C 180,E1 -10868.72,E2 -10868.72} C_VEL
LIN {X 0,Y 406.25,Z 340.749,A -85,B 0,C 180,E1 -10869.793,E2 -10869.793} C_VEL
LIN {X 0,Y 410.44,Z 364.407,A -85,B 0,C 180,E1 -10870.489,E2 -10870.489} C_VEL
LIN {X 0,Y 411.198,Z 371.411,A -85,B 0,C 180,E1 -10870.663,E2 -10870.663} C_VEL
LIN {X 0,Y 410.023,Z 450.194,A -85,B 0,C 180,E1 -10872.096,E2 -10872.096} C_VEL
LIN {X 0,Y 409.412,Z 463.854,A -85,B 0,C 180,E1 -10872.552,E2 -10872.552} C_VEL
LIN {X 0,Y 408.691,Z 475.631,A -85,B 0,C 180,E1 -10873.132,E2 -10873.132} C_VEL
LIN {X 0,Y 407.833,Z 486.815,A -85,B 0,C 180,E1 -10873.868,E2 -10873.868} C_VEL
LIN {X 0,Y 406.908,Z 498.412,A -85,B 0,C 180,E1 -10874.858,E2 -10874.858} C_VEL
LIN {X 0,Y 405.929,Z 508.868,A -85,B 0,C 180,E1 -10875.974,E2 -10875.974} C_VEL
LIN {X 0,Y 405.21,Z 518.311,A -85,B 0,C 180,E1 -10877.226,E2 -10877.226} C_VEL
LIN {X 0,Y 404.321,Z 527.428,A -85,B 0,C 180,E1 -10878.725,E2 -10878.725} C_VEL
LIN {X 0,Y 403.7,Z 534.793,A -85,B 0,C 180,E1 -10880.229,E2 -10880.229} C_VEL
LIN {X 0,Y 403.248,Z 541.584,A -85,B 0,C 180,E1 -10881.987,E2 -10881.987} C_VEL
LIN {X 0,Y 402.937,Z 546.908,A -85,B 0,C 180,E1 -10883.823,E2 -10883.823} C_VEL
LIN {X 0,Y 402.93,Z 549.512,A -85,B 0,C 180,E1 -10884.998,E2 -10884.998} C_VEL
LIN {X 0,Y 402.827,Z 552.532,A -85,B 0,C 180,E1 -10887.001,E2 -10887.001} C_VEL
LIN {X 0,Y 402.907,Z 553.452,A -85,B 0,C 180,E1 -10888.002,E2 -10888.002} C_VEL
LIN {X 0,Y 402.866,Z 553.95,A -85,B 0,C 180,E1 -10889.002,E2 -10889.002} C_VEL
LIN {X 0,Y 402.871,Z 554.031,A -85,B 0,C 180,E1 -10890.001,E2 -10890.001} C_VEL
LIN {X 0,Y 402.912,Z 553.034,A -85,B 0,C 180,E1 -10892.001,E2 -10892.001} C_VEL
LIN {X 0,Y 402.859,Z 551.92,A -85,B 0,C 180,E1 -10893.001,E2 -10893.001} C_VEL
LIN {X 0,Y 402.858,Z 550.361,A -85,B 0,C 180,E1 -10894.003,E2 -10894.003} C_VEL
LIN {X 0,Y 402.917,Z 547.223,A -85,B 0,C 180,E1 -10895.507,E2 -10895.507} C_VEL
LIN {X 0,Y 403.077,Z 543.011,A -85,B 0,C 180,E1 -10897.012,E2 -10897.012} C_VEL
LIN {X 0,Y 403.374,Z 536.582,A -85,B 0,C 180,E1 -10898.77,E2 -10898.77} C_VEL
LIN {X 0,Y 403.766,Z 529.561,A -85,B 0,C 180,E1 -10900.279,E2 -10900.279} C_VEL
LIN {X 0,Y 404.384,Z 520.748,A -85,B 0,C 180,E1 -10901.785,E2 -10901.785} C_VEL
LIN {X 0,Y 405.057,Z 511.715,A -85,B 0,C 180,E1 -10903.037,E2 -10903.037} C_VEL
LIN {X 0,Y 405.743,Z 501.771,A -85,B 0,C 180,E1 -10904.163,E2 -10904.163} C_VEL
LIN {X 0,Y 406.433,Z 490.755,A -85,B 0,C 180,E1 -10905.163,E2 -10905.163} C_VEL
LIN {X 0,Y 407.201,Z 478.395,A -85,B 0,C 180,E1 -10906.032,E2 -10906.032} C_VEL
LIN {X 0,Y 407.93,Z 465.353,A -85,B 0,C 180,E1 -10906.71,E2 -10906.71} C_VEL
LIN {X 0,Y 408.468,Z 452.074,A -85,B 0,C 180,E1 -10907.17,E2 -10907.17} C_VEL
LIN {X 0,Y 408.813,Z 431.466,A -85,B 0,C 180,E1 -10907.574,E2 -10907.574} C_VEL
LIN {X 0,Y 409.39,Z 368.308,A -85,B 0,C 180,E1 -10908.689,E2 -10908.689} C_VEL
LIN {X 0,Y 405.472,Z 341.194,A -85,B 0,C 180,E1 -10909.361,E2 -10909.361} C_VEL
LIN {X 0,Y 406.418,Z 325.988,A -85,B 0,C 180,E1 -10912.362,E2 -10912.362} C_VEL
LIN {X 0,Y 407.07,Z 315.353,A -85,B 0,C 180,E1 -10914.48,E2 -10914.48} C_VEL
LIN {X 0,Y 405.102,Z 304.47,A -85,B 0,C 180,E1 -10916.813,E2 -10916.813} C_VEL
LIN {X 0,Y 404.253,Z 300.132,A -85,B 0,C 180,E1 -10917.795,E2 -10917.795} C_VEL
LIN {X 0,Y 404.145,Z 300.139,A -85,B 0,C 180,E1 -10921.559,E2 -10921.559} C_VEL
LIN {X 0,Y 404.19,Z 300.133,A -85,B 0,C 180,E1 -10925.017,E2 -10925.017} C_VEL
LIN {X 0,Y 404.155,Z 300.141,A -85,B 0,C 180,E1 -10928.758,E2 -10928.758} C_VEL
LIN {X 0,Y 404.129,Z 300.14,A -85,B 0,C 180,E1 -10931.6,E2 -10931.6} C_VEL
LIN {X 0,Y 404.151,Z 300.144,A -85,B 0,C 180,E1 -10934.522,E2 -10934.522} C_VEL
LIN {X 0,Y 404.143,Z 300.14,A -85,B 0,C 180,E1 -10937.296,E2 -10937.296} C_VEL
LIN {X 0,Y 404.176,Z 300.135,A -85,B 0,C 180,E1 -10939.956,E2 -10939.956} C_VEL
LIN {X 0,Y 404.142,Z 300.143,A -85,B 0,C 180,E1 -10943.125,E2 -10943.125} C_VEL
LIN {X 0,Y 404.144,Z 300.139,A -85,B 0,C 180,E1 -10946.187,E2 -10946.187} C_VEL
LIN {X 0,Y 404.152,Z 300.139,A -85,B 0,C 180,E1 -10949.715,E2 -10949.715} C_VEL
LIN {X 0,Y 404.202,Z 300.138,A -85,B 0,C 180,E1 -10953.123,E2 -10953.123} C_VEL
LIN {X 0,Y 404.181,Z 300.141,A -85,B 0,C 180,E1 -10955.334,E2 -10955.334} C_VEL
LIN {X 0,Y 404.145,Z 300.138,A -85,B 0,C 180,E1 -10958.581,E2 -10958.581} C_VEL
LIN {X 0,Y 404.211,Z 300.134,A -85,B 0,C 180,E1 -10961.762,E2 -10961.762} C_VEL
LIN {X 0,Y 404.212,Z 300.13,A -85,B 0,C 180,E1 -10964.882,E2 -10964.882} C_VEL
LIN {X 0,Y 404.261,Z 300.128,A -85,B 0,C 180,E1 -10967.958,E2 -10967.958} C_VEL
LIN {X 0,Y 404.282,Z 300.121,A -85,B 0,C 180,E1 -10970.999,E2 -10970.999} C_VEL
LIN {X 0,Y 404.39,Z 300.114,A -85,B 0,C 180,E1 -10974.014,E2 -10974.014} C_VEL
LIN {X 0,Y 404.486,Z 300.103,A -85,B 0,C 180,E1 -10978.008,E2 -10978.008} C_VEL
LIN {X 0,Y 404.613,Z 300.086,A -85,B 0,C 180,E1 -10980,E2 -10980} C_VEL
LIN {X 0,Y 404.419,Z 300.104,A -85,B 0,C 180,E1 -10982.988,E2 -10982.988} C_VEL
LIN {X 0,Y 404.386,Z 300.108,A -85,B 0,C 180,E1 -10986.628,E2 -10986.628} C_VEL
LIN {X 0,Y 404.262,Z 300.126,A -85,B 0,C 180,E1 -10990.011,E2 -10990.011} C_VEL
LIN {X 0,Y 404.272,Z 300.123,A -85,B 0,C 180,E1 -10993.211,E2 -10993.211} C_VEL
LIN {X 0,Y 404.221,Z 300.132,A -85,B 0,C 180,E1 -10997.006,E2 -10997.006} C_VEL
LIN {X 0,Y 404.169,Z 300.138,A -85,B 0,C 180,E1 -11000.351,E2 -11000.351} C_VEL
LIN {X 0,Y 404.169,Z 300.136,A -85,B 0,C 180,E1 -11003.574,E2 -11003.574} C_VEL
LIN {X 0,Y 404.189,Z 300.133,A -85,B 0,C 180,E1 -11005.766,E2 -11005.766} C_VEL
LIN {X 0,Y 404.2,Z 300.131,A -85,B 0,C 180,E1 -11007.999,E2 -11007.999} C_VEL
LIN {X 0,Y 404.144,Z 300.141,A -85,B 0,C 180,E1 -11011.557,E2 -11011.557} C_VEL
LIN {X 0,Y 404.189,Z 300.137,A -85,B 0,C 180,E1 -11015.016,E2 -11015.016} C_VEL
LIN {X 0,Y 404.16,Z 300.137,A -85,B 0,C 180,E1 -11018.756,E2 -11018.756} C_VEL
LIN {X 0,Y 404.128,Z 300.147,A -85,B 0,C 180,E1 -11021.599,E2 -11021.599} C_VEL
LIN {X 0,Y 404.149,Z 300.138,A -85,B 0,C 180,E1 -11024.521,E2 -11024.521} C_VEL
LIN {X 0,Y 404.14,Z 300.142,A -85,B 0,C 180,E1 -11027.295,E2 -11027.295} C_VEL
LIN {X 0,Y 404.173,Z 300.14,A -85,B 0,C 180,E1 -11029.955,E2 -11029.955} C_VEL
LIN {X 0,Y 404.139,Z 300.139,A -85,B 0,C 180,E1 -11033.124,E2 -11033.124} C_VEL
LIN {X 0,Y 404.149,Z 300.142,A -85,B 0,C 180,E1 -11036.187,E2 -11036.187} C_VEL
LIN {X 0,Y 404.149,Z 300.141,A -85,B 0,C 180,E1 -11039.714,E2 -11039.714} C_VEL
LIN {X 0,Y 404.198,Z 300.132,A -85,B 0,C 180,E1 -11043.122,E2 -11043.122} C_VEL
LIN {X 0,Y 404.18,Z 300.134,A -85,B 0,C 180,E1 -11045.333,E2 -11045.333} C_VEL
LIN {X 0,Y 404.166,Z 300.14,A -85,B 0,C 180,E1 -11048.581,E2 -11048.581} C_VEL
LIN {X 0,Y 404.216,Z 300.13,A -85,B 0,C 180,E1 -11051.761,E2 -11051.761} C_VEL
LIN {X 0,Y 404.209,Z 300.134,A -85,B 0,C 180,E1 -11054.881,E2 -11054.881} C_VEL
LIN {X 0,Y 404.258,Z 300.125,A -85,B 0,C 180,E1 -11057.957,E2 -11057.957} C_VEL
LIN {X 0,Y 404.267,Z 300.131,A -85,B 0,C 180,E1 -11060.997,E2 -11060.997} C_VEL
LIN {X 0,Y 404.349,Z 300.145,A -85,B 0,C 180,E1 -11062.74,E2 -11062.74} C_VEL
LIN {X 0,Y 405.794,Z 308.781,A -85,B 0,C 180,E1 -11064.782,E2 -11064.782} C_VEL
LIN {X 0,Y 405.796,Z 313.072,A -85,B 0,C 180,E1 -11065.746,E2 -11065.746} C_VEL
LIN {X 0,Y 409.83,Z 334.16,A -85,B 0,C 180,E1 -11066.301,E2 -11066.301} C_VEL
LIN {X 0,Y 408.677,Z 420.845,A -85,B 0,C 180,E1 -11067.847,E2 -11067.847} C_VEL
LIN {X 0,Y 408.233,Z 433.884,A -85,B 0,C 180,E1 -11068.276,E2 -11068.276} C_VEL
LIN {X 0,Y 407.842,Z 446.431,A -85,B 0,C 180,E1 -11068.895,E2 -11068.895} C_VEL
LIN {X 0,Y 407.155,Z 459.184,A -85,B 0,C 180,E1 -11069.757,E2 -11069.757} C_VEL
LIN {X 0,Y 406.41,Z 470.446,A -85,B 0,C 180,E1 -11070.742,E2 -11070.742} C_VEL
LIN {X 0,Y 405.619,Z 480.68,A -85,B 0,C 180,E1 -11071.86,E2 -11071.86} C_VEL
LIN {X 0,Y 405.392,Z 484.022,A -85,B 0,C 180,E1 -11072.289,E2 -11072.289} C_VEL
LIN {X 0,Y 404.475,Z 488.281,A -85,B 0,C 180,E1 -11072.856,E2 -11072.856} C_VEL
LIN {X 0,Y 401.196,Z 494.837,A -85,B 0,C 180,E1 -11073.804,E2 -11073.804} C_VEL
LIN {X 0,Y 397.862,Z 500.825,A -85,B 0,C 180,E1 -11074.835,E2 -11074.835} C_VEL
LIN {X 0,Y 396.874,Z 504.147,A -85,B 0,C 180,E1 -11075.527,E2 -11075.527} C_VEL
LIN {X 0,Y 396.546,Z 510.508,A -85,B 0,C 180,E1 -11077.125,E2 -11077.125} C_VEL
LIN {X 0,Y 396.177,Z 515.363,A -85,B 0,C 180,E1 -11078.671,E2 -11078.671} C_VEL
LIN {X 0,Y 395.949,Z 519.087,A -85,B 0,C 180,E1 -11080.222,E2 -11080.222} C_VEL
LIN {X 0,Y 395.861,Z 521.011,A -85,B 0,C 180,E1 -11081.26,E2 -11081.26} C_VEL
LIN {X 0,Y 395.761,Z 522.567,A -85,B 0,C 180,E1 -11082.393,E2 -11082.393} C_VEL
LIN {X 0,Y 395.658,Z 524.128,A -85,B 0,C 180,E1 -11084.398,E2 -11084.398} C_VEL
LIN {X 0,Y 395.685,Z 524.342,A -85,B 0,C 180,E1 -11085.45,E2 -11085.45} C_VEL
LIN {X 0,Y 395.669,Z 524.102,A -85,B 0,C 180,E1 -11086.509,E2 -11086.509} C_VEL
LIN {X 0,Y 395.746,Z 523.452,A -85,B 0,C 180,E1 -11087.57,E2 -11087.57} C_VEL
LIN {X 0,Y 395.834,Z 522.388,A -85,B 0,C 180,E1 -11088.636,E2 -11088.636} C_VEL
LIN {X 0,Y 396.027,Z 520.571,A -85,B 0,C 180,E1 -11089.856,E2 -11089.856} C_VEL
LIN {X 0,Y 396.362,Z 516.321,A -85,B 0,C 180,E1 -11091.859,E2 -11091.859} C_VEL
LIN {X 0,Y 396.81,Z 511.498,A -85,B 0,C 180,E1 -11093.483,E2 -11093.483} C_VEL
LIN {X 0,Y 397.447,Z 505.27,A -85,B 0,C 180,E1 -11095.11,E2 -11095.11} C_VEL
LIN {X 0,Y 398.254,Z 497.401,A -85,B 0,C 180,E1 -11096.742,E2 -11096.742} C_VEL
LIN {X 0,Y 399.131,Z 488.538,A -85,B 0,C 180,E1 -11098.205,E2 -11098.205} C_VEL
LIN {X 0,Y 400.057,Z 479.092,A -85,B 0,C 180,E1 -11099.463,E2 -11099.463} C_VEL
LIN {X 0,Y 401.065,Z 468.003,A -85,B 0,C 180,E1 -11100.651,E2 -11100.651} C_VEL
LIN {X 0,Y 402.023,Z 456.288,A -85,B 0,C 180,E1 -11101.629,E2 -11101.629} C_VEL
LIN {X 0,Y 402.709,Z 444.703,A -85,B 0,C 180,E1 -11102.379,E2 -11102.379} C_VEL
LIN {X 0,Y 403.393,Z 431.591,A -85,B 0,C 180,E1 -11102.996,E2 -11102.996} C_VEL
LIN {X 0,Y 403.772,Z 418.766,A -85,B 0,C 180,E1 -11103.383,E2 -11103.383} C_VEL
LIN {X 0,Y 405.133,Z 335.702,A -85,B 0,C 180,E1 -11104.896,E2 -11104.896} C_VEL
LIN {X 0,Y 400.99,Z 317.657,A -85,B 0,C 180,E1 -11105.5,E2 -11105.5} C_VEL
LIN {X 0,Y 399.666,Z 313.336,A -85,B 0,C 180,E1 -11105.696,E2 -11105.696} C_VEL
LIN {X 0,Y 397.077,Z 301.023,A -85,B 0,C 180,E1 -11108.751,E2 -11108.751} C_VEL
LIN {X 0,Y 397.043,Z 301.029,A -85,B 0,C 180,E1 -11112.268,E2 -11112.268} C_VEL
LIN {X 0,Y 397.075,Z 301.026,A -85,B 0,C 180,E1 -11115.068,E2 -11115.068} C_VEL
LIN {X 0,Y 397.041,Z 301.028,A -85,B 0,C 180,E1 -11118.022,E2 -11118.022} C_VEL
LIN {X 0,Y 397.077,Z 301.028,A -85,B 0,C 180,E1 -11121.722,E2 -11121.722} C_VEL
LIN {X 0,Y 397.109,Z 301.009,A -85,B 0,C 180,E1 -11125.505,E2 -11125.505} C_VEL
LIN {X 0,Y 397.064,Z 301.02,A -85,B 0,C 180,E1 -11129.116,E2 -11129.116} C_VEL
LIN {X 0,Y 397.088,Z 301.019,A -85,B 0,C 180,E1 -11132.602,E2 -11132.602} C_VEL
LIN {X 0,Y 397.106,Z 301.018,A -85,B 0,C 180,E1 -11135.98,E2 -11135.98} C_VEL
LIN {X 0,Y 397.125,Z 301.011,A -85,B 0,C 180,E1 -11139.704,E2 -11139.704} C_VEL
LIN {X 0,Y 397.168,Z 301.004,A -85,B 0,C 180,E1 -11142.844,E2 -11142.844} C_VEL
LIN {X 0,Y 397.214,Z 301.001,A -85,B 0,C 180,E1 -11146.702,E2 -11146.702} C_VEL
LIN {X 0,Y 397.209,Z 301.004,A -85,B 0,C 180,E1 -11149.809,E2 -11149.809} C_VEL
LIN {X 0,Y 397.302,Z 300.985,A -85,B 0,C 180,E1 -11152.887,E2 -11152.887} C_VEL
LIN {X 0,Y 397.232,Z 301.002,A -85,B 0,C 180,E1 -11154.925,E2 -11154.925} C_VEL
LIN {X 0,Y 397.435,Z 300.971,A -85,B 0,C 180,E1 -11157.973,E2 -11157.973} C_VEL
LIN {X 0,Y 397.565,Z 300.958,A -85,B 0,C 180,E1 -11160,E2 -11160} C_VEL
LIN {X 0,Y 397.361,Z 300.976,A -85,B 0,C 180,E1 -11163.042,E2 -11163.042} C_VEL
LIN {X 0,Y 397.348,Z 300.984,A -85,B 0,C 180,E1 -11167.112,E2 -11167.112} C_VEL
LIN {X 0,Y 397.205,Z 301.002,A -85,B 0,C 180,E1 -11170.192,E2 -11170.192} C_VEL
LIN {X 0,Y 397.213,Z 300.995,A -85,B 0,C 180,E1 -11173.322,E2 -11173.322} C_VEL
LIN {X 0,Y 397.169,Z 301.009,A -85,B 0,C 180,E1 -11177.156,E2 -11177.156} C_VEL
LIN {X 0,Y 397.09,Z 301.02,A -85,B 0,C 180,E1 -11180.731,E2 -11180.731} C_VEL
LIN {X 0,Y 397.12,Z 301.009,A -85,B 0,C 180,E1 -11184.019,E2 -11184.019} C_VEL
LIN {X 0,Y 397.183,Z 301.004,A -85,B 0,C 180,E1 -11187.391,E2 -11187.391} C_VEL
LIN {X 0,Y 397.078,Z 301.024,A -85,B 0,C 180,E1 -11190.883,E2 -11190.883} C_VEL
LIN {X 0,Y 397.116,Z 301.018,A -85,B 0,C 180,E1 -11194.495,E2 -11194.495} C_VEL
LIN {X 0,Y 397.1,Z 301.019,A -85,B 0,C 180,E1 -11198.276,E2 -11198.276} C_VEL
LIN {X 0,Y 397.105,Z 301.021,A -85,B 0,C 180,E1 -11200.907,E2 -11200.907} C_VEL
LIN {X 0,Y 397.098,Z 301.023,A -85,B 0,C 180,E1 -11203.649,E2 -11203.649} C_VEL
LIN {X 0,Y 397.152,Z 301.005,A -85,B 0,C 180,E1 -11206.514,E2 -11206.514} C_VEL
LIN {X 0,Y 397.116,Z 301.013,A -85,B 0,C 180,E1 -11209.553,E2 -11209.553} C_VEL
LIN {X 0,Y 397.093,Z 301.02,A -85,B 0,C 180,E1 -11212.792,E2 -11212.792} C_VEL
LIN {X 0,Y 397.113,Z 301.015,A -85,B 0,C 180,E1 -11216.284,E2 -11216.284} C_VEL
LIN {X 0,Y 397.101,Z 301.02,A -85,B 0,C 180,E1 -11220.137,E2 -11220.137} C_VEL
LIN {X 0,Y 397.165,Z 301.129,A -85,B 0,C 180,E1 -11220.738,E2 -11220.738} C_VEL
LIN {X 0,Y 399.947,Z 313.381,A -85,B 0,C 180,E1 -11223.662,E2 -11223.662} C_VEL
LIN {X 0,Y 401.029,Z 319.846,A -85,B 0,C 180,E1 -11225.13,E2 -11225.13} C_VEL
LIN {X 0,Y 399.787,Z 335.405,A -85,B 0,C 180,E1 -11228.338,E2 -11228.338} C_VEL
LIN {X 0,Y 399.415,Z 340.455,A -85,B 0,C 180,E1 -11229.369,E2 -11229.369} C_VEL
LIN {X 0,Y 403.9,Z 365.321,A -85,B 0,C 180,E1 -11230.125,E2 -11230.125} C_VEL
LIN {X 0,Y 404.63,Z 372.408,A -85,B 0,C 180,E1 -11230.303,E2 -11230.303} C_VEL
LIN {X 0,Y 403.379,Z 449.579,A -85,B 0,C 180,E1 -11231.725,E2 -11231.725} C_VEL
LIN {X 0,Y 402.763,Z 463.334,A -85,B 0,C 180,E1 -11232.189,E2 -11232.189} C_VEL
LIN {X 0,Y 401.928,Z 476.229,A -85,B 0,C 180,E1 -11232.84,E2 -11232.84} C_VEL
LIN {X 0,Y 400.903,Z 488.754,A -85,B 0,C 180,E1 -11233.713,E2 -11233.713} C_VEL
LIN {X 0,Y 399.964,Z 499.935,A -85,B 0,C 180,E1 -11234.72,E2 -11234.72} C_VEL
LIN {X 0,Y 398.969,Z 509.98,A -85,B 0,C 180,E1 -11235.847,E2 -11235.847} C_VEL
LIN {X 0,Y 398.134,Z 519.983,A -85,B 0,C 180,E1 -11237.254,E2 -11237.254} C_VEL
LIN {X 0,Y 397.162,Z 528.77,A -85,B 0,C 180,E1 -11238.777,E2 -11238.777} C_VEL
LIN {X 0,Y 396.602,Z 535.817,A -85,B 0,C 180,E1 -11240.31,E2 -11240.31} C_VEL
LIN {X 0,Y 396.196,Z 541.468,A -85,B 0,C 180,E1 -11241.843,E2 -11241.843} C_VEL
LIN {X 0,Y 395.928,Z 546.057,A -85,B 0,C 180,E1 -11243.427,E2 -11243.427} C_VEL
LIN {X 0,Y 395.842,Z 549.329,A -85,B 0,C 180,E1 -11244.909,E2 -11244.909} C_VEL
LIN {X 0,Y 395.775,Z 551.024,A -85,B 0,C 180,E1 -11245.928,E2 -11245.928} C_VEL
LIN {X 0,Y 395.803,Z 553.222,A -85,B 0,C 180,E1 -11247.966,E2 -11247.966} C_VEL
LIN {X 0,Y 395.795,Z 553.693,A -85,B 0,C 180,E1 -11248.984,E2 -11248.984} C_VEL
LIN {X 0,Y 395.797,Z 553.759,A -85,B 0,C 180,E1 -11250.002,E2 -11250.002} C_VEL
LIN {X 0,Y 395.811,Z 553.44,A -85,B 0,C 180,E1 -11251.019,E2 -11251.019} C_VEL
LIN {X 0,Y 395.826,Z 552.732,A -85,B 0,C 180,E1 -11252.037,E2 -11252.037} C_VEL
LIN {X 0,Y 395.76,Z 551.588,A -85,B 0,C 180,E1 -11253.055,E2 -11253.055} C_VEL
LIN {X 0,Y 395.781,Z 550.013,A -85,B 0,C 180,E1 -11254.075,E2 -11254.075} C_VEL
LIN {X 0,Y 395.829,Z 546.345,A -85,B 0,C 180,E1 -11255.806,E2 -11255.806} C_VEL
LIN {X 0,Y 396.06,Z 540.939,A -85,B 0,C 180,E1 -11257.649,E2 -11257.649} C_VEL
LIN {X 0,Y 396.437,Z 533.913,A -85,B 0,C 180,E1 -11259.44,E2 -11259.44} C_VEL
LIN {X 0,Y 396.885,Z 526.297,A -85,B 0,C 180,E1 -11260.975,E2 -11260.975} C_VEL
LIN {X 0,Y 397.558,Z 518.523,A -85,B 0,C 180,E1 -11262.249,E2 -11262.249} C_VEL
LIN {X 0,Y 398.254,Z 509.53,A -85,B 0,C 180,E1 -11263.462,E2 -11263.462} C_VEL
LIN {X 0,Y 398.978,Z 498.443,A -85,B 0,C 180,E1 -11264.669,E2 -11264.669} C_VEL
LIN {X 0,Y 399.787,Z 486.681,A -85,B 0,C 180,E1 -11265.682,E2 -11265.682} C_VEL
LIN {X 0,Y 400.577,Z 474.112,A -85,B 0,C 180,E1 -11266.501,E2 -11266.501} C_VEL
LIN {X 0,Y 401.251,Z 460.847,A -85,B 0,C 180,E1 -11267.127,E2 -11267.127} C_VEL
LIN {X 0,Y 401.715,Z 448.864,A -85,B 0,C 180,E1 -11267.501,E2 -11267.501} C_VEL
LIN {X 0,Y 402.584,Z 369.197,A -85,B 0,C 180,E1 -11268.946,E2 -11268.946} C_VEL
LIN {X 0,Y 398.526,Z 340.989,A -85,B 0,C 180,E1 -11269.645,E2 -11269.645} C_VEL
LIN {X 0,Y 399.629,Z 324.113,A -85,B 0,C 180,E1 -11273.036,E2 -11273.036} C_VEL
LIN {X 0,Y 400.053,Z 316.109,A -85,B 0,C 180,E1 -11274.665,E2 -11274.665} C_VEL
LIN {X 0,Y 397.764,Z 303.838,A -85,B 0,C 180,E1 -11277.349,E2 -11277.349} C_VEL
LIN {X 0,Y 397.208,Z 301.009,A -85,B 0,C 180,E1 -11278.009,E2 -11278.009} C_VEL
LIN {X 0,Y 397.088,Z 301.021,A -85,B 0,C 180,E1 -11281.837,E2 -11281.837} C_VEL
LIN {X 0,Y 397.131,Z 301.017,A -85,B 0,C 180,E1 -11284.494,E2 -11284.494} C_VEL
LIN {X 0,Y 397.105,Z 301.021,A -85,B 0,C 180,E1 -11288.276,E2 -11288.276} C_VEL
LIN {X 0,Y 397.095,Z 301.019,A -85,B 0,C 180,E1 -11290.909,E2 -11290.909} C_VEL
LIN {X 0,Y 397.107,Z 301.015,A -85,B 0,C 180,E1 -11293.649,E2 -11293.649} C_VEL
LIN {X 0,Y 397.109,Z 301.021,A -85,B 0,C 180,E1 -11296.521,E2 -11296.521} C_VEL
LIN {X 0,Y 397.12,Z 301.016,A -85,B 0,C 180,E1 -11300.423,E2 -11300.423} C_VEL
LIN {X 0,Y 397.112,Z 301.015,A -85,B 0,C 180,E1 -11304.265,E2 -11304.265} C_VEL
LIN {X 0,Y 397.118,Z 301.018,A -85,B 0,C 180,E1 -11306.727,E2 -11306.727} C_VEL
LIN {X 0,Y 397.131,Z 301.012,A -85,B 0,C 180,E1 -11310.296,E2 -11310.296} C_VEL
LIN {X 0,Y 397.201,Z 301.005,A -85,B 0,C 180,E1 -11312.61,E2 -11312.61} C_VEL
LIN {X 0,Y 397.135,Z 301.012,A -85,B 0,C 180,E1 -11315.982,E2 -11315.982} C_VEL
LIN {X 0,Y 397.145,Z 301.014,A -85,B 0,C 180,E1 -11319.705,E2 -11319.705} C_VEL
LIN {X 0,Y 397.188,Z 301.006,A -85,B 0,C 180,E1 -11322.845,E2 -11322.845} C_VEL
LIN {X 0,Y 397.235,Z 300.999,A -85,B 0,C 180,E1 -11326.703,E2 -11326.703} C_VEL
LIN {X 0,Y 397.223,Z 301.008,A -85,B 0,C 180,E1 -11329.809,E2 -11329.809} C_VEL
LIN {X 0,Y 397.302,Z 300.991,A -85,B 0,C 180,E1 -11332.887,E2 -11332.887} C_VEL
LIN {X 0,Y 397.25,Z 300.997,A -85,B 0,C 180,E1 -11334.925,E2 -11334.925} C_VEL
LIN {X 0,Y 397.455,Z 300.979,A -85,B 0,C 180,E1 -11337.973,E2 -11337.973} C_VEL
LIN {X 0,Y 397.582,Z 300.962,A -85,B 0,C 180,E1 -11340,E2 -11340} C_VEL
LIN {X 0,Y 397.379,Z 300.981,A -85,B 0,C 180,E1 -11343.041,E2 -11343.041} C_VEL
LIN {X 0,Y 397.337,Z 300.987,A -85,B 0,C 180,E1 -11346.624,E2 -11346.624} C_VEL
LIN {X 0,Y 397.241,Z 300.999,A -85,B 0,C 180,E1 -11349.162,E2 -11349.162} C_VEL
LIN {X 0,Y 397.224,Z 301.005,A -85,B 0,C 180,E1 -11352.258,E2 -11352.258} C_VEL
LIN {X 0,Y 397.185,Z 301.006,A -85,B 0,C 180,E1 -11355.392,E2 -11355.392} C_VEL
LIN {X 0,Y 397.163,Z 301.014,A -85,B 0,C 180,E1 -11358.573,E2 -11358.573} C_VEL
LIN {X 0,Y 397.101,Z 301.016,A -85,B 0,C 180,E1 -11361.818,E2 -11361.818} C_VEL
LIN {X 0,Y 397.158,Z 301.01,A -85,B 0,C 180,E1 -11365.512,E2 -11365.512} C_VEL
LIN {X 0,Y 397.127,Z 301.014,A -85,B 0,C 180,E1 -11368.543,E2 -11368.543} C_VEL
LIN {X 0,Y 397.083,Z 301.018,A -85,B 0,C 180,E1 -11372.071,E2 -11372.071} C_VEL
LIN {X 0,Y 397.123,Z 301.018,A -85,B 0,C 180,E1 -11375.502,E2 -11375.502} C_VEL
LIN {X 0,Y 397.135,Z 301.013,A -85,B 0,C 180,E1 -11378.861,E2 -11378.861} C_VEL
LIN {X 0,Y 397.073,Z 301.02,A -85,B 0,C 180,E1 -11382.266,E2 -11382.266} C_VEL
LIN {X 0,Y 397.091,Z 301.019,A -85,B 0,C 180,E1 -11385.068,E2 -11385.068} C_VEL
LIN {X 0,Y 397.07,Z 301.023,A -85,B 0,C 180,E1 -11388.02,E2 -11388.02} C_VEL
LIN {X 0,Y 397.13,Z 301.013,A -85,B 0,C 180,E1 -11391.138,E2 -11391.138} C_VEL
LIN {X 0,Y 397.123,Z 301.014,A -85,B 0,C 180,E1 -11394.496,E2 -11394.496} C_VEL
LIN {X 0,Y 397.083,Z 301.025,A -85,B 0,C 180,E1 -11397.927,E2 -11397.927} C_VEL
LIN {X 0,Y 397.125,Z 301.014,A -85,B 0,C 180,E1 -11401.455,E2 -11401.455} C_VEL
LIN {X 0,Y 397.156,Z 301.013,A -85,B 0,C 180,E1 -11404.487,E2 -11404.487} C_VEL
LIN {X 0,Y 397.114,Z 301.02,A -85,B 0,C 180,E1 -11408.181,E2 -11408.181} C_VEL
LIN {X 0,Y 397.174,Z 301.007,A -85,B 0,C 180,E1 -11411.426,E2 -11411.426} C_VEL
LIN {X 0,Y 397.182,Z 301.013,A -85,B 0,C 180,E1 -11414.607,E2 -11414.607} C_VEL
LIN {X 0,Y 397.221,Z 301.001,A -85,B 0,C 180,E1 -11417.741,E2 -11417.741} C_VEL
LIN {X 0,Y 397.237,Z 301.007,A -85,B 0,C 180,E1 -11420.836,E2 -11420.836} C_VEL
LIN {X 0,Y 397.318,Z 301.012,A -85,B 0,C 180,E1 -11422.537,E2 -11422.537} C_VEL
LIN {X 0,Y 398.812,Z 309.964,A -85,B 0,C 180,E1 -11424.69,E2 -11424.69} C_VEL
LIN {X 0,Y 398.821,Z 313.287,A -85,B 0,C 180,E1 -11425.451,E2 -11425.451} C_VEL
LIN {X 0,Y 403.052,Z 335.067,A -85,B 0,C 180,E1 -11426.036,E2 -11426.036} C_VEL
LIN {X 0,Y 401.822,Z 420.81,A -85,B 0,C 180,E1 -11427.586,E2 -11427.586} C_VEL
LIN {X 0,Y 401.361,Z 433.999,A -85,B 0,C 180,E1 -11428.025,E2 -11428.025} C_VEL
LIN {X 0,Y 400.946,Z 446.933,A -85,B 0,C 180,E1 -11428.674,E2 -11428.674} C_VEL
LIN {X 0,Y 400.328,Z 458.296,A -85,B 0,C 180,E1 -11429.445,E2 -11429.445} C_VEL
LIN {X 0,Y 399.49,Z 470.347,A -85,B 0,C 180,E1 -11430.502,E2 -11430.502} C_VEL
LIN {X 0,Y 398.685,Z 480.65,A -85,B 0,C 180,E1 -11431.64,E2 -11431.64} C_VEL
LIN {X 0,Y 398.081,Z 489.052,A -85,B 0,C 180,E1 -11432.781,E2 -11432.781} C_VEL
LIN {X 0,Y 397.33,Z 498.182,A -85,B 0,C 180,E1 -11434.31,E2 -11434.31} C_VEL
LIN {X 0,Y 396.874,Z 504.147,A -85,B 0,C 180,E1 -11435.527,E2 -11435.527} C_VEL
LIN {X 0,Y 395.928,Z 507.275,A -85,B 0,C 180,E1 -11436.244,E2 -11436.244} C_VEL
LIN {X 0,Y 392.783,Z 511.897,A -85,B 0,C 180,E1 -11437.435,E2 -11437.435} C_VEL
LIN {X 0,Y 389.741,Z 515.846,A -85,B 0,C 180,E1 -11438.692,E2 -11438.692} C_VEL
LIN {X 0,Y 388.97,Z 517.867,A -85,B 0,C 180,E1 -11439.503,E2 -11439.503} C_VEL
LIN {X 0,Y 388.836,Z 519.819,A -85,B 0,C 180,E1 -11440.411,E2 -11440.411} C_VEL
LIN {X 0,Y 388.741,Z 521.619,A -85,B 0,C 180,E1 -11441.469,E2 -11441.469} C_VEL
LIN {X 0,Y 388.659,Z 522.981,A -85,B 0,C 180,E1 -11442.531,E2 -11442.531} C_VEL
LIN {X 0,Y 388.588,Z 523.941,A -85,B 0,C 180,E1 -11443.597,E2 -11443.597} C_VEL
LIN {X 0,Y 388.56,Z 524.486,A -85,B 0,C 180,E1 -11444.666,E2 -11444.666} C_VEL
LIN {X 0,Y 388.591,Z 524.381,A -85,B 0,C 180,E1 -11446.555,E2 -11446.555} C_VEL
LIN {X 0,Y 388.698,Z 523.542,A -85,B 0,C 180,E1 -11447.899,E2 -11447.899} C_VEL
LIN {X 0,Y 388.798,Z 522.347,A -85,B 0,C 180,E1 -11448.986,E2 -11448.986} C_VEL
LIN {X 0,Y 389.062,Z 519.714,A -85,B 0,C 180,E1 -11450.623,E2 -11450.623} C_VEL
LIN {X 0,Y 389.406,Z 515.96,A -85,B 0,C 180,E1 -11452.27,E2 -11452.27} C_VEL
LIN {X 0,Y 389.907,Z 510.959,A -85,B 0,C 180,E1 -11453.924,E2 -11453.924} C_VEL
LIN {X 0,Y 390.605,Z 504.544,A -85,B 0,C 180,E1 -11455.581,E2 -11455.581} C_VEL
LIN {X 0,Y 391.332,Z 497.892,A -85,B 0,C 180,E1 -11456.964,E2 -11456.964} C_VEL
LIN {X 0,Y 392.132,Z 490.331,A -85,B 0,C 180,E1 -11458.262,E2 -11458.262} C_VEL
LIN {X 0,Y 393.132,Z 480.853,A -85,B 0,C 180,E1 -11459.592,E2 -11459.592} C_VEL
LIN {X 0,Y 394.18,Z 469.744,A -85,B 0,C 180,E1 -11460.835,E2 -11460.835} C_VEL
LIN {X 0,Y 395.1,Z 459.404,A -85,B 0,C 180,E1 -11461.756,E2 -11461.756} C_VEL
LIN {X 0,Y 395.871,Z 448.106,A -85,B 0,C 180,E1 -11462.555,E2 -11462.555} C_VEL
LIN {X 0,Y 396.614,Z 435.599,A -85,B 0,C 180,E1 -11463.204,E2 -11463.204} C_VEL
LIN {X 0,Y 397.106,Z 421.855,A -85,B 0,C 180,E1 -11463.687,E2 -11463.687} C_VEL
LIN {X 0,Y 398.523,Z 336.296,A -85,B 0,C 180,E1 -11465.294,E2 -11465.294} C_VEL
LIN {X 0,Y 394.469,Z 318.973,A -85,B 0,C 180,E1 -11465.897,E2 -11465.897} C_VEL
LIN {X 0,Y 392.57,Z 313.676,A -85,B 0,C 180,E1 -11466.144,E2 -11466.144} C_VEL
LIN {X 0,Y 390.017,Z 301.902,A -85,B 0,C 180,E1 -11469.154,E2 -11469.154} C_VEL
LIN {X 0,Y 390.018,Z 301.904,A -85,B 0,C 180,E1 -11472.37,E2 -11472.37} C_VEL
LIN {X 0,Y 390.032,Z 301.899,A -85,B 0,C 180,E1 -11475.353,E2 -11475.353} C_VEL
LIN {X 0,Y 390.004,Z 301.904,A -85,B 0,C 180,E1 -11478.183,E2 -11478.183} C_VEL
LIN {X 0,Y 390.044,Z 301.899,A -85,B 0,C 180,E1 -11480.902,E2 -11480.902} C_VEL
LIN {X 0,Y 390.059,Z 301.882,A -85,B 0,C 180,E1 -11484.791,E2 -11484.791} C_VEL
LIN {X 0,Y 390.009,Z 301.898,A -85,B 0,C 180,E1 -11488.495,E2 -11488.495} C_VEL
LIN {X 0,Y 390.025,Z 301.9,A -85,B 0,C 180,E1 -11492.063,E2 -11492.063} C_VEL
LIN {X 0,Y 390.038,Z 301.895,A -85,B 0,C 180,E1 -11495.517,E2 -11495.517} C_VEL
LIN {X 0,Y 390.041,Z 301.891,A -85,B 0,C 180,E1 -11498.877,E2 -11498.877} C_VEL
LIN {X 0,Y 390.113,Z 301.888,A -85,B 0,C 180,E1 -11502.166,E2 -11502.166} C_VEL
LIN {X 0,Y 390.129,Z 301.886,A -85,B 0,C 180,E1 -11505.392,E2 -11505.392} C_VEL
LIN {X 0,Y 390.133,Z 301.883,A -85,B 0,C 180,E1 -11508.571,E2 -11508.571} C_VEL
LIN {X 0,Y 390.248,Z 301.871,A -85,B 0,C 180,E1 -11512.079,E2 -11512.079} C_VEL
LIN {X 0,Y 390.202,Z 301.879,A -85,B 0,C 180,E1 -11514.833,E2 -11514.833} C_VEL
LIN {X 0,Y 390.404,Z 301.847,A -85,B 0,C 180,E1 -11517.937,E2 -11517.937} C_VEL
LIN {X 0,Y 390.535,Z 301.834,A -85,B 0,C 180,E1 -11520,E2 -11520} C_VEL
LIN {X 0,Y 390.296,Z 301.856,A -85,B 0,C 180,E1 -11523.097,E2 -11523.097} C_VEL
LIN {X 0,Y 390.313,Z 301.864,A -85,B 0,C 180,E1 -11526.202,E2 -11526.202} C_VEL
LIN {X 0,Y 390.301,Z 301.86,A -85,B 0,C 180,E1 -11528.283,E2 -11528.283} C_VEL
LIN {X 0,Y 390.158,Z 301.884,A -85,B 0,C 180,E1 -11532.484,E2 -11532.484} C_VEL
LIN {X 0,Y 390.126,Z 301.886,A -85,B 0,C 180,E1 -11535.678,E2 -11535.678} C_VEL
LIN {X 0,Y 390.092,Z 301.886,A -85,B 0,C 180,E1 -11538.923,E2 -11538.923} C_VEL
LIN {X 0,Y 390.027,Z 301.898,A -85,B 0,C 180,E1 -11542.235,E2 -11542.235} C_VEL
LIN {X 0,Y 390.107,Z 301.89,A -85,B 0,C 180,E1 -11545.745,E2 -11545.745} C_VEL
LIN {X 0,Y 390.055,Z 301.895,A -85,B 0,C 180,E1 -11549.11,E2 -11549.11} C_VEL
LIN {X 0,Y 390.045,Z 301.893,A -85,B 0,C 180,E1 -11552.722,E2 -11552.722} C_VEL
LIN {X 0,Y 390.047,Z 301.896,A -85,B 0,C 180,E1 -11555.827,E2 -11555.827} C_VEL
LIN {X 0,Y 390.065,Z 301.896,A -85,B 0,C 180,E1 -11559.221,E2 -11559.221} C_VEL
LIN {X 0,Y 390.073,Z 301.892,A -85,B 0,C 180,E1 -11562.382,E2 -11562.382} C_VEL
LIN {X 0,Y 390.095,Z 301.882,A -85,B 0,C 180,E1 -11566.108,E2 -11566.108} C_VEL
LIN {X 0,Y 390.076,Z 301.894,A -85,B 0,C 180,E1 -11569.176,E2 -11569.176} C_VEL
LIN {X 0,Y 390.041,Z 301.9,A -85,B 0,C 180,E1 -11572.45,E2 -11572.45} C_VEL
LIN {X 0,Y 390.063,Z 301.894,A -85,B 0,C 180,E1 -11576.047,E2 -11576.047} C_VEL
LIN {X 0,Y 390.042,Z 301.901,A -85,B 0,C 180,E1 -11579.871,E2 -11579.871} C_VEL
LIN {X 0,Y 390.107,Z 302.009,A -85,B 0,C 180,E1 -11580.341,E2 -11580.341} C_VEL
LIN {X 0,Y 392.746,Z 313.439,A -85,B 0,C 180,E1 -11583.141,E2 -11583.141} C_VEL
LIN {X 0,Y 394.105,Z 321.006,A -85,B 0,C 180,E1 -11584.906,E2 -11584.906} C_VEL
LIN {X 0,Y 393.44,Z 330.252,A -85,B 0,C 180,E1 -11586.862,E2 -11586.862} C_VEL
LIN {X 0,Y 392.578,Z 340.181,A -85,B 0,C 180,E1 -11588.928,E2 -11588.928} C_VEL
LIN {X 0,Y 396.863,Z 363.046,A -85,B 0,C 180,E1 -11589.655,E2 -11589.655} C_VEL
LIN {X 0,Y 398.085,Z 372.316,A -85,B 0,C 180,E1 -11589.911,E2 -11589.911} C_VEL
LIN {X 0,Y 396.777,Z 449.188,A -85,B 0,C 180,E1 -11591.349,E2 -11591.349} C_VEL
LIN {X 0,Y 396.164,Z 462.847,A -85,B 0,C 180,E1 -11591.815,E2 -11591.815} C_VEL
LIN {X 0,Y 395.375,Z 474.73,A -85,B 0,C 180,E1 -11592.413,E2 -11592.413} C_VEL
LIN {X 0,Y 394.401,Z 486.005,A -85,B 0,C 180,E1 -11593.17,E2 -11593.17} C_VEL
LIN {X 0,Y 393.354,Z 497.645,A -85,B 0,C 180,E1 -11594.191,E2 -11594.191} C_VEL
LIN {X 0,Y 392.202,Z 508.502,A -85,B 0,C 180,E1 -11595.386,E2 -11595.386} C_VEL
LIN {X 0,Y 391.373,Z 518.429,A -85,B 0,C 180,E1 -11596.766,E2 -11596.766} C_VEL
LIN {X 0,Y 390.347,Z 527.422,A -85,B 0,C 180,E1 -11598.316,E2 -11598.316} C_VEL
LIN {X 0,Y 389.657,Z 534.687,A -85,B 0,C 180,E1 -11599.873,E2 -11599.873} C_VEL
LIN {X 0,Y 389.135,Z 541.354,A -85,B 0,C 180,E1 -11601.694,E2 -11601.694} C_VEL
LIN {X 0,Y 388.851,Z 545.781,A -85,B 0,C 180,E1 -11603.255,E2 -11603.255} C_VEL
LIN {X 0,Y 388.739,Z 549.146,A -85,B 0,C 180,E1 -11604.815,E2 -11604.815} C_VEL
LIN {X 0,Y 388.7,Z 550.827,A -85,B 0,C 180,E1 -11605.854,E2 -11605.854} C_VEL
LIN {X 0,Y 388.7,Z 552.989,A -85,B 0,C 180,E1 -11607.929,E2 -11607.929} C_VEL
LIN {X 0,Y 388.726,Z 553.435,A -85,B 0,C 180,E1 -11608.966,E2 -11608.966} C_VEL
LIN {X 0,Y 388.726,Z 553.487,A -85,B 0,C 180,E1 -11610.002,E2 -11610.002} C_VEL
LIN {X 0,Y 388.741,Z 553.153,A -85,B 0,C 180,E1 -11611.037,E2 -11611.037} C_VEL
LIN {X 0,Y 388.725,Z 552.427,A -85,B 0,C 180,E1 -11612.074,E2 -11612.074} C_VEL
LIN {X 0,Y 388.665,Z 551.253,A -85,B 0,C 180,E1 -11613.111,E2 -11613.111} C_VEL
LIN {X 0,Y 388.721,Z 548.727,A -85,B 0,C 180,E1 -11614.668,E2 -11614.668} C_VEL
LIN {X 0,Y 388.796,Z 545.174,A -85,B 0,C 180,E1 -11616.228,E2 -11616.228} C_VEL
LIN {X 0,Y 388.994,Z 540.499,A -85,B 0,C 180,E1 -11617.789,E2 -11617.789} C_VEL
LIN {X 0,Y 389.388,Z 533.431,A -85,B 0,C 180,E1 -11619.612,E2 -11619.612} C_VEL
LIN {X 0,Y 389.876,Z 525.768,A -85,B 0,C 180,E1 -11621.175,E2 -11621.175} C_VEL
LIN {X 0,Y 390.556,Z 517.928,A -85,B 0,C 180,E1 -11622.472,E2 -11622.472} C_VEL
LIN {X 0,Y 391.388,Z 507.704,A -85,B 0,C 180,E1 -11623.843,E2 -11623.843} C_VEL
LIN {X 0,Y 392.066,Z 497.665,A -85,B 0,C 180,E1 -11624.934,E2 -11624.934} C_VEL
LIN {X 0,Y 392.893,Z 485.729,A -85,B 0,C 180,E1 -11625.965,E2 -11625.965} C_VEL
LIN {X 0,Y 393.698,Z 472.919,A -85,B 0,C 180,E1 -11626.798,E2 -11626.798} C_VEL
LIN {X 0,Y 394.415,Z 460.095,A -85,B 0,C 180,E1 -11627.4,E2 -11627.4} C_VEL
LIN {X 0,Y 394.843,Z 447.645,A -85,B 0,C 180,E1 -11627.782,E2 -11627.782} C_VEL
LIN {X 0,Y 395.832,Z 370.698,A -85,B 0,C 180,E1 -11629.192,E2 -11629.192} C_VEL
LIN {X 0,Y 391.553,Z 340.766,A -85,B 0,C 180,E1 -11629.941,E2 -11629.941} C_VEL
LIN {X 0,Y 392.542,Z 326.208,A -85,B 0,C 180,E1 -11632.919,E2 -11632.919} C_VEL
LIN {X 0,Y 393.144,Z 318.231,A -85,B 0,C 180,E1 -11634.56,E2 -11634.56} C_VEL
LIN {X 0,Y 391.848,Z 310.496,A -85,B 0,C 180,E1 -11636.262,E2 -11636.262} C_VEL
LIN {X 0,Y 390.183,Z 301.884,A -85,B 0,C 180,E1 -11638.227,E2 -11638.227} C_VEL
LIN {X 0,Y 390.038,Z 301.902,A -85,B 0,C 180,E1 -11642.125,E2 -11642.125} C_VEL
LIN {X 0,Y 390.091,Z 301.889,A -85,B 0,C 180,E1 -11645.208,E2 -11645.208} C_VEL
LIN {X 0,Y 390.072,Z 301.892,A -85,B 0,C 180,E1 -11649.218,E2 -11649.218} C_VEL
LIN {X 0,Y 390.048,Z 301.9,A -85,B 0,C 180,E1 -11652.375,E2 -11652.375} C_VEL
LIN {X 0,Y 390.05,Z 301.895,A -85,B 0,C 180,E1 -11655.355,E2 -11655.355} C_VEL
LIN {X 0,Y 390.037,Z 301.897,A -85,B 0,C 180,E1 -11658.187,E2 -11658.187} C_VEL
LIN {X 0,Y 390.095,Z 301.895,A -85,B 0,C 180,E1 -11660.908,E2 -11660.908} C_VEL
LIN {X 0,Y 390.088,Z 301.895,A -85,B 0,C 180,E1 -11664.793,E2 -11664.793} C_VEL
LIN {X 0,Y 390.029,Z 301.898,A -85,B 0,C 180,E1 -11668.496,E2 -11668.496} C_VEL
LIN {X 0,Y 390.124,Z 301.885,A -85,B 0,C 180,E1 -11672.07,E2 -11672.07} C_VEL
LIN {X 0,Y 390.084,Z 301.895,A -85,B 0,C 180,E1 -11675.519,E2 -11675.519} C_VEL
LIN {X 0,Y 390.094,Z 301.895,A -85,B 0,C 180,E1 -11679.53,E2 -11679.53} C_VEL
LIN {X 0,Y 390.144,Z 301.886,A -85,B 0,C 180,E1 -11683.248,E2 -11683.248} C_VEL
LIN {X 0,Y 390.201,Z 301.875,A -85,B 0,C 180,E1 -11686.562,E2 -11686.562} C_VEL
LIN {X 0,Y 390.173,Z 301.885,A -85,B 0,C 180,E1 -11689.623,E2 -11689.623} C_VEL
LIN {X 0,Y 390.255,Z 301.869,A -85,B 0,C 180,E1 -11692.758,E2 -11692.758} C_VEL
LIN {X 0,Y 390.22,Z 301.873,A -85,B 0,C 180,E1 -11694.833,E2 -11694.833} C_VEL
LIN {X 0,Y 390.423,Z 301.854,A -85,B 0,C 180,E1 -11697.937,E2 -11697.937} C_VEL
LIN {X 0,Y 390.552,Z 301.838,A -85,B 0,C 180,E1 -11700,E2 -11700} C_VEL
LIN {X 0,Y 390.313,Z 301.861,A -85,B 0,C 180,E1 -11703.096,E2 -11703.096} C_VEL
LIN {X 0,Y 390.292,Z 301.866,A -85,B 0,C 180,E1 -11706.617,E2 -11706.617} C_VEL
LIN {X 0,Y 390.199,Z 301.876,A -85,B 0,C 180,E1 -11709.329,E2 -11709.329} C_VEL
LIN {X 0,Y 390.176,Z 301.886,A -85,B 0,C 180,E1 -11712.483,E2 -11712.483} C_VEL
LIN {X 0,Y 390.145,Z 301.882,A -85,B 0,C 180,E1 -11715.676,E2 -11715.676} C_VEL
LIN {X 0,Y 390.108,Z 301.892,A -85,B 0,C 180,E1 -11718.922,E2 -11718.922} C_VEL
LIN {X 0,Y 390.043,Z 301.896,A -85,B 0,C 180,E1 -11722.234,E2 -11722.234} C_VEL
LIN {X 0,Y 390.125,Z 301.885,A -85,B 0,C 180,E1 -11725.743,E2 -11725.743} C_VEL
LIN {X 0,Y 390.064,Z 301.899,A -85,B 0,C 180,E1 -11729.109,E2 -11729.109} C_VEL
LIN {X 0,Y 390.048,Z 301.897,A -85,B 0,C 180,E1 -11732.721,E2 -11732.721} C_VEL
LIN {X 0,Y 390.06,Z 301.894,A -85,B 0,C 180,E1 -11735.824,E2 -11735.824} C_VEL
LIN {X 0,Y 390.075,Z 301.896,A -85,B 0,C 180,E1 -11739.218,E2 -11739.218} C_VEL
LIN {X 0,Y 390.047,Z 301.895,A -85,B 0,C 180,E1 -11742.373,E2 -11742.373} C_VEL
LIN {X 0,Y 390.048,Z 301.899,A -85,B 0,C 180,E1 -11745.353,E2 -11745.353} C_VEL
LIN {X 0,Y 390.035,Z 301.898,A -85,B 0,C 180,E1 -11748.186,E2 -11748.186} C_VEL
LIN {X 0,Y 390.091,Z 301.889,A -85,B 0,C 180,E1 -11750.906,E2 -11750.906} C_VEL
LIN {X 0,Y 390.089,Z 301.889,A -85,B 0,C 180,E1 -11754.792,E2 -11754.792} C_VEL
LIN {X 0,Y 390.027,Z 301.899,A -85,B 0,C 180,E1 -11758.495,E2 -11758.495} C_VEL
LIN {X 0,Y 390.121,Z 301.892,A -85,B 0,C 180,E1 -11762.069,E2 -11762.069} C_VEL
LIN {X 0,Y 390.082,Z 301.891,A -85,B 0,C 180,E1 -11765.518,E2 -11765.518} C_VEL
LIN {X 0,Y 390.075,Z 301.893,A -85,B 0,C 180,E1 -11768.878,E2 -11768.878} C_VEL
LIN {X 0,Y 390.133,Z 301.887,A -85,B 0,C 180,E1 -11772.166,E2 -11772.166} C_VEL
LIN {X 0,Y 390.146,Z 301.882,A -85,B 0,C 180,E1 -11775.391,E2 -11775.391} C_VEL
LIN {X 0,Y 390.15,Z 301.888,A -85,B 0,C 180,E1 -11778.57,E2 -11778.57} C_VEL
LIN {X 0,Y 390.319,Z 302.052,A -85,B 0,C 180,E1 -11782.371,E2 -11782.371} C_VEL
LIN {X 0,Y 391.854,Z 311.172,A -85,B 0,C 180,E1 -11784.596,E2 -11784.596} C_VEL
LIN {X 0,Y 391.907,Z 313.827,A -85,B 0,C 180,E1 -11785.16,E2 -11785.16} C_VEL
LIN {X 0,Y 396.248,Z 336.005,A -85,B 0,C 180,E1 -11785.768,E2 -11785.768} C_VEL
LIN {X 0,Y 394.975,Z 420.728,A -85,B 0,C 180,E1 -11787.321,E2 -11787.321} C_VEL
LIN {X 0,Y 394.514,Z 433.979,A -85,B 0,C 180,E1 -11787.765,E2 -11787.765} C_VEL
LIN {X 0,Y 394.079,Z 446.443,A -85,B 0,C 180,E1 -11788.393,E2 -11788.393} C_VEL
LIN {X 0,Y 393.398,Z 458.695,A -85,B 0,C 180,E1 -11789.231,E2 -11789.231} C_VEL
LIN {X 0,Y 392.581,Z 470.208,A -85,B 0,C 180,E1 -11790.255,E2 -11790.255} C_VEL
LIN {X 0,Y 391.742,Z 480.589,A -85,B 0,C 180,E1 -11791.412,E2 -11791.412} C_VEL
LIN {X 0,Y 391.122,Z 489.052,A -85,B 0,C 180,E1 -11792.573,E2 -11792.573} C_VEL
LIN {X 0,Y 390.311,Z 498.25,A -85,B 0,C 180,E1 -11794.129,E2 -11794.129} C_VEL
LIN {X 0,Y 389.74,Z 505.641,A -85,B 0,C 180,E1 -11795.69,E2 -11795.69} C_VEL
LIN {X 0,Y 389.444,Z 511.554,A -85,B 0,C 180,E1 -11797.256,E2 -11797.256} C_VEL
LIN {X 0,Y 389.08,Z 516.246,A -85,B 0,C 180,E1 -11798.83,E2 -11798.83} C_VEL
LIN {X 0,Y 388.97,Z 517.867,A -85,B 0,C 180,E1 -11799.503,E2 -11799.503} C_VEL
LIN {X 0,Y 388.2,Z 519.673,A -85,B 0,C 180,E1 -11800.326,E2 -11800.326} C_VEL
LIN {X 0,Y 385.202,Z 522.16,A -85,B 0,C 180,E1 -11801.679,E2 -11801.679} C_VEL
LIN {X 0,Y 382.693,Z 523.588,A -85,B 0,C 180,E1 -11802.789,E2 -11802.789} C_VEL
LIN {X 0,Y 381.588,Z 524.267,A -85,B 0,C 180,E1 -11803.659,E2 -11803.659} C_VEL
LIN {X 0,Y 381.483,Z 524.406,A -85,B 0,C 180,E1 -11803.955,E2 -11803.955} C_VEL
LIN {X 0,Y 381.488,Z 524.811,A -85,B 0,C 180,E1 -11806.04,E2 -11806.04} C_VEL
LIN {X 0,Y 381.53,Z 524.429,A -85,B 0,C 180,E1 -11807.139,E2 -11807.139} C_VEL
LIN {X 0,Y 381.641,Z 523.587,A -85,B 0,C 180,E1 -11808.242,E2 -11808.242} C_VEL
LIN {X 0,Y 381.933,Z 521.002,A -85,B 0,C 180,E1 -11810.206,E2 -11810.206} C_VEL
LIN {X 0,Y 382.308,Z 517.062,A -85,B 0,C 180,E1 -11812.137,E2 -11812.137} C_VEL
LIN {X 0,Y 382.802,Z 512.322,A -85,B 0,C 180,E1 -11813.821,E2 -11813.821} C_VEL
LIN {X 0,Y 383.512,Z 506.171,A -85,B 0,C 180,E1 -11815.506,E2 -11815.506} C_VEL
LIN {X 0,Y 384.436,Z 498.387,A -85,B 0,C 180,E1 -11817.194,E2 -11817.194} C_VEL
LIN {X 0,Y 385.402,Z 489.8,A -85,B 0,C 180,E1 -11818.687,E2 -11818.687} C_VEL
LIN {X 0,Y 386.428,Z 480.344,A -85,B 0,C 180,E1 -11820.007,E2 -11820.007} C_VEL
LIN {X 0,Y 387.427,Z 470.463,A -85,B 0,C 180,E1 -11821.129,E2 -11821.129} C_VEL
LIN {X 0,Y 388.435,Z 459.766,A -85,B 0,C 180,E1 -11822.104,E2 -11822.104} C_VEL
LIN {X 0,Y 389.275,Z 448.029,A -85,B 0,C 180,E1 -11822.946,E2 -11822.946} C_VEL
LIN {X 0,Y 390.045,Z 435.379,A -85,B 0,C 180,E1 -11823.605,E2 -11823.605} C_VEL
LIN {X 0,Y 390.537,Z 421.883,A -85,B 0,C 180,E1 -11824.083,E2 -11824.083} C_VEL
LIN {X 0,Y 392.107,Z 337.844,A -85,B 0,C 180,E1 -11825.678,E2 -11825.678} C_VEL
LIN {X 0,Y 388.351,Z 321.609,A -85,B 0,C 180,E1 -11826.256,E2 -11826.256} C_VEL
LIN {X 0,Y 385.397,Z 313.918,A -85,B 0,C 180,E1 -11826.643,E2 -11826.643} C_VEL
LIN {X 0,Y 382.97,Z 302.782,A -85,B 0,C 180,E1 -11829.578,E2 -11829.578} C_VEL
LIN {X 0,Y 382.995,Z 302.779,A -85,B 0,C 180,E1 -11832.777,E2 -11832.777} C_VEL
LIN {X 0,Y 382.984,Z 302.772,A -85,B 0,C 180,E1 -11835.787,E2 -11835.787} C_VEL
LIN {X 0,Y 382.95,Z 302.783,A -85,B 0,C 180,E1 -11838.799,E2 -11838.799} C_VEL
LIN {X 0,Y 382.979,Z 302.781,A -85,B 0,C 180,E1 -11842.097,E2 -11842.097} C_VEL
LIN {X 0,Y 382.999,Z 302.764,A -85,B 0,C 180,E1 -11845.33,E2 -11845.33} C_VEL
LIN {X 0,Y 382.969,Z 302.775,A -85,B 0,C 180,E1 -11849.08,E2 -11849.08} C_VEL
LIN {X 0,Y 382.979,Z 302.777,A -85,B 0,C 180,E1 -11852.692,E2 -11852.692} C_VEL
LIN {X 0,Y 383,Z 302.777,A -85,B 0,C 180,E1 -11856.191,E2 -11856.191} C_VEL
LIN {X 0,Y 383.041,Z 302.764,A -85,B 0,C 180,E1 -11859.598,E2 -11859.598} C_VEL
LIN {X 0,Y 383.091,Z 302.757,A -85,B 0,C 180,E1 -11862.931,E2 -11862.931} C_VEL
LIN {X 0,Y 383.111,Z 302.76,A -85,B 0,C 180,E1 -11866.464,E2 -11866.464} C_VEL
LIN {X 0,Y 383.139,Z 302.76,A -85,B 0,C 180,E1 -11870.498,E2 -11870.498} C_VEL
LIN {X 0,Y 383.24,Z 302.736,A -85,B 0,C 180,E1 -11873.683,E2 -11873.683} C_VEL
LIN {X 0,Y 383.371,Z 302.722,A -85,B 0,C 180,E1 -11877.899,E2 -11877.899} C_VEL
LIN {X 0,Y 383.504,Z 302.709,A -85,B 0,C 180,E1 -11880,E2 -11880} C_VEL
LIN {X 0,Y 383.232,Z 302.735,A -85,B 0,C 180,E1 -11883.154,E2 -11883.154} C_VEL
LIN {X 0,Y 383.271,Z 302.742,A -85,B 0,C 180,E1 -11886.317,E2 -11886.317} C_VEL
LIN {X 0,Y 383.246,Z 302.737,A -85,B 0,C 180,E1 -11888.436,E2 -11888.436} C_VEL
LIN {X 0,Y 383.084,Z 302.762,A -85,B 0,C 180,E1 -11891.643,E2 -11891.643} C_VEL
LIN {X 0,Y 383.096,Z 302.76,A -85,B 0,C 180,E1 -11894.883,E2 -11894.883} C_VEL
LIN {X 0,Y 383.076,Z 302.761,A -85,B 0,C 180,E1 -11898.173,E2 -11898.173} C_VEL
LIN {X 0,Y 382.98,Z 302.777,A -85,B 0,C 180,E1 -11901.532,E2 -11901.532} C_VEL
LIN {X 0,Y 383.04,Z 302.769,A -85,B 0,C 180,E1 -11904.961,E2 -11904.961} C_VEL
LIN {X 0,Y 383.038,Z 302.763,A -85,B 0,C 180,E1 -11908.493,E2 -11908.493} C_VEL
LIN {X 0,Y 383.027,Z 302.766,A -85,B 0,C 180,E1 -11912.148,E2 -11912.148} C_VEL
LIN {X 0,Y 383.017,Z 302.772,A -85,B 0,C 180,E1 -11915.957,E2 -11915.957} C_VEL
LIN {X 0,Y 383.013,Z 302.775,A -85,B 0,C 180,E1 -11919.589,E2 -11919.589} C_VEL
LIN {X 0,Y 383.024,Z 302.771,A -85,B 0,C 180,E1 -11922.785,E2 -11922.785} C_VEL
LIN {X 0,Y 383.031,Z 302.761,A -85,B 0,C 180,E1 -11925.797,E2 -11925.797} C_VEL
LIN {X 0,Y 383.037,Z 302.771,A -85,B 0,C 180,E1 -11928.788,E2 -11928.788} C_VEL
LIN {X 0,Y 382.997,Z 302.78,A -85,B 0,C 180,E1 -11932.097,E2 -11932.097} C_VEL
LIN {X 0,Y 383.013,Z 302.779,A -85,B 0,C 180,E1 -11935.334,E2 -11935.334} C_VEL
LIN {X 0,Y 382.978,Z 302.777,A -85,B 0,C 180,E1 -11939.083,E2 -11939.083} C_VEL
LIN {X 0,Y 383.023,Z 302.896,A -85,B 0,C 180,E1 -11939.921,E2 -11939.921} C_VEL
LIN {X 0,Y 385.558,Z 313.516,A -85,B 0,C 180,E1 -11942.598,E2 -11942.598} C_VEL
LIN {X 0,Y 387.23,Z 322.537,A -85,B 0,C 180,E1 -11944.756,E2 -11944.756} C_VEL
LIN {X 0,Y 386.681,Z 330.3,A -85,B 0,C 180,E1 -11946.433,E2 -11946.433} C_VEL
LIN {X 0,Y 385.789,Z 339.92,A -85,B 0,C 180,E1 -11948.47,E2 -11948.47} C_VEL
LIN {X 0,Y 389.888,Z 361.4,A -85,B 0,C 180,E1 -11949.177,E2 -11949.177} C_VEL
LIN {X 0,Y 391.559,Z 372.919,A -85,B 0,C 180,E1 -11949.514,E2 -11949.514} C_VEL
LIN {X 0,Y 390.197,Z 448.745,A -85,B 0,C 180,E1 -11950.956,E2 -11950.956} C_VEL
LIN {X 0,Y 389.563,Z 462.397,A -85,B 0,C 180,E1 -11951.428,E2 -11951.428} C_VEL
LIN {X 0,Y 388.707,Z 474.318,A -85,B 0,C 180,E1 -11952.033,E2 -11952.033} C_VEL
LIN {X 0,Y 387.643,Z 486.418,A -85,B 0,C 180,E1 -11952.867,E2 -11952.867} C_VEL
LIN {X 0,Y 386.545,Z 497.928,A -85,B 0,C 180,E1 -11953.905,E2 -11953.905} C_VEL
LIN {X 0,Y 385.394,Z 508.318,A -85,B 0,C 180,E1 -11955.075,E2 -11955.075} C_VEL
LIN {X 0,Y 384.66,Z 516.827,A -85,B 0,C 180,E1 -11956.262,E2 -11956.262} C_VEL
LIN {X 0,Y 383.754,Z 524.701,A -85,B 0,C 180,E1 -11957.575,E2 -11957.575} C_VEL
LIN {X 0,Y 382.846,Z 532.419,A -85,B 0,C 180,E1 -11959.156,E2 -11959.156} C_VEL
LIN {X 0,Y 382.219,Z 539.544,A -85,B 0,C 180,E1 -11961.01,E2 -11961.01} C_VEL
LIN {X 0,Y 381.865,Z 544.309,A -85,B 0,C 180,E1 -11962.6,E2 -11962.6} C_VEL
LIN {X 0,Y 381.694,Z 547.331,A -85,B 0,C 180,E1 -11963.873,E2 -11963.873} C_VEL
LIN {X 0,Y 381.625,Z 550.634,A -85,B 0,C 180,E1 -11965.777,E2 -11965.777} C_VEL
LIN {X 0,Y 381.598,Z 552.753,A -85,B 0,C 180,E1 -11967.891,E2 -11967.891} C_VEL
LIN {X 0,Y 381.639,Z 553.178,A -85,B 0,C 180,E1 -11968.946,E2 -11968.946} C_VEL
LIN {X 0,Y 381.656,Z 553.215,A -85,B 0,C 180,E1 -11970.002,E2 -11970.002} C_VEL
LIN {X 0,Y 381.672,Z 552.865,A -85,B 0,C 180,E1 -11971.057,E2 -11971.057} C_VEL
LIN {X 0,Y 381.624,Z 552.115,A -85,B 0,C 180,E1 -11972.112,E2 -11972.112} C_VEL
LIN {X 0,Y 381.632,Z 549.311,A -85,B 0,C 180,E1 -11974.226,E2 -11974.226} C_VEL
LIN {X 0,Y 381.69,Z 545.338,A -85,B 0,C 180,E1 -11976.121,E2 -11976.121} C_VEL
LIN {X 0,Y 381.919,Z 540.048,A -85,B 0,C 180,E1 -11977.934,E2 -11977.934} C_VEL
LIN {X 0,Y 382.332,Z 532.931,A -85,B 0,C 180,E1 -11979.791,E2 -11979.791} C_VEL
LIN {X 0,Y 382.885,Z 525.203,A -85,B 0,C 180,E1 -11981.382,E2 -11981.382} C_VEL
LIN {X 0,Y 383.557,Z 517.28,A -85,B 0,C 180,E1 -11982.703,E2 -11982.703} C_VEL
LIN {X 0,Y 384.37,Z 507.931,A -85,B 0,C 180,E1 -11983.98,E2 -11983.98} C_VEL
LIN {X 0,Y 385.156,Z 496.827,A -85,B 0,C 180,E1 -11985.208,E2 -11985.208} C_VEL
LIN {X 0,Y 385.902,Z 486.41,A -85,B 0,C 180,E1 -11986.126,E2 -11986.126} C_VEL
LIN {X 0,Y 386.73,Z 473.928,A -85,B 0,C 180,E1 -11986.973,E2 -11986.973} C_VEL
LIN {X 0,Y 387.5,Z 460.784,A -85,B 0,C 180,E1 -11987.619,E2 -11987.619} C_VEL
LIN {X 0,Y 387.983,Z 447.743,A -85,B 0,C 180,E1 -11988.039,E2 -11988.039} C_VEL
LIN {X 0,Y 389.007,Z 371.887,A -85,B 0,C 180,E1 -11989.455,E2 -11989.455} C_VEL
LIN {X 0,Y 384.632,Z 340.398,A -85,B 0,C 180,E1 -11990.275,E2 -11990.275} C_VEL
LIN {X 0,Y 385.894,Z 323.266,A -85,B 0,C 180,E1 -11993.843,E2 -11993.843} C_VEL
LIN {X 0,Y 386.153,Z 318.97,A -85,B 0,C 180,E1 -11994.748,E2 -11994.748} C_VEL
LIN {X 0,Y 384.153,Z 308.04,A -85,B 0,C 180,E1 -11997.219,E2 -11997.219} C_VEL
LIN {X 0,Y 383.116,Z 302.765,A -85,B 0,C 180,E1 -11998.488,E2 -11998.488} C_VEL
LIN {X 0,Y 382.993,Z 302.778,A -85,B 0,C 180,E1 -12002.423,E2 -12002.423} C_VEL
LIN {X 0,Y 383.031,Z 302.772,A -85,B 0,C 180,E1 -12005.956,E2 -12005.956} C_VEL
LIN {X 0,Y 383.019,Z 302.77,A -85,B 0,C 180,E1 -12009.587,E2 -12009.587} C_VEL
LIN {X 0,Y 383.012,Z 302.776,A -85,B 0,C 180,E1 -12012.779,E2 -12012.779} C_VEL
LIN {X 0,Y 383.003,Z 302.772,A -85,B 0,C 180,E1 -12015.79,E2 -12015.79} C_VEL
LIN {X 0,Y 382.995,Z 302.78,A -85,B 0,C 180,E1 -12018.796,E2 -12018.796} C_VEL
LIN {X 0,Y 383.005,Z 302.772,A -85,B 0,C 180,E1 -12022.097,E2 -12022.097} C_VEL
LIN {X 0,Y 383.023,Z 302.773,A -85,B 0,C 180,E1 -12025.332,E2 -12025.332} C_VEL
LIN {X 0,Y 382.989,Z 302.781,A -85,B 0,C 180,E1 -12029.082,E2 -12029.082} C_VEL
LIN {X 0,Y 383.063,Z 302.766,A -85,B 0,C 180,E1 -12032.698,E2 -12032.698} C_VEL
LIN {X 0,Y 383.058,Z 302.77,A -85,B 0,C 180,E1 -12035.04,E2 -12035.04} C_VEL
LIN {X 0,Y 382.999,Z 302.773,A -85,B 0,C 180,E1 -12038.469,E2 -12038.469} C_VEL
LIN {X 0,Y 383.059,Z 302.769,A -85,B 0,C 180,E1 -12041.826,E2 -12041.826} C_VEL
LIN {X 0,Y 383.116,Z 302.76,A -85,B 0,C 180,E1 -12045.118,E2 -12045.118} C_VEL
LIN {X 0,Y 383.102,Z 302.761,A -85,B 0,C 180,E1 -12048.358,E2 -12048.358} C_VEL
LIN {X 0,Y 383.222,Z 302.75,A -85,B 0,C 180,E1 -12052.027,E2 -12052.027} C_VEL
LIN {X 0,Y 383.19,Z 302.749,A -85,B 0,C 180,E1 -12054.738,E2 -12054.738} C_VEL
LIN {X 0,Y 383.391,Z 302.729,A -85,B 0,C 180,E1 -12057.899,E2 -12057.899} C_VEL
LIN {X 0,Y 383.521,Z 302.714,A -85,B 0,C 180,E1 -12060,E2 -12060} C_VEL
LIN {X 0,Y 383.249,Z 302.741,A -85,B 0,C 180,E1 -12063.153,E2 -12063.153} C_VEL
LIN {X 0,Y 383.252,Z 302.745,A -85,B 0,C 180,E1 -12066.607,E2 -12066.607} C_VEL
LIN {X 0,Y 383.149,Z 302.754,A -85,B 0,C 180,E1 -12069.502,E2 -12069.502} C_VEL
LIN {X 0,Y 383.131,Z 302.756,A -85,B 0,C 180,E1 -12073.536,E2 -12073.536} C_VEL
LIN {X 0,Y 383.1,Z 302.763,A -85,B 0,C 180,E1 -12077.069,E2 -12077.069} C_VEL
LIN {X 0,Y 383.034,Z 302.774,A -85,B 0,C 180,E1 -12080.646,E2 -12080.646} C_VEL
LIN {X 0,Y 383.031,Z 302.768,A -85,B 0,C 180,E1 -12083.807,E2 -12083.807} C_VEL
LIN {X 0,Y 383.085,Z 302.762,A -85,B 0,C 180,E1 -12086.123,E2 -12086.123} C_VEL
LIN {X 0,Y 382.997,Z 302.774,A -85,B 0,C 180,E1 -12089.699,E2 -12089.699} C_VEL
LIN {X 0,Y 383.008,Z 302.776,A -85,B 0,C 180,E1 -12093.4,E2 -12093.4} C_VEL
LIN {X 0,Y 383.036,Z 302.768,A -85,B 0,C 180,E1 -12096.164,E2 -12096.164} C_VEL
LIN {X 0,Y 383.013,Z 302.772,A -85,B 0,C 180,E1 -12099.958,E2 -12099.958} C_VEL
LIN {X 0,Y 383.01,Z 302.772,A -85,B 0,C 180,E1 -12102.778,E2 -12102.778} C_VEL
LIN {X 0,Y 383.001,Z 302.777,A -85,B 0,C 180,E1 -12105.788,E2 -12105.788} C_VEL
LIN {X 0,Y 382.992,Z 302.773,A -85,B 0,C 180,E1 -12108.795,E2 -12108.795} C_VEL
LIN {X 0,Y 383.002,Z 302.776,A -85,B 0,C 180,E1 -12112.096,E2 -12112.096} C_VEL
LIN {X 0,Y 383.022,Z 302.771,A -85,B 0,C 180,E1 -12115.331,E2 -12115.331} C_VEL
LIN {X 0,Y 382.987,Z 302.774,A -85,B 0,C 180,E1 -12119.08,E2 -12119.08} C_VEL
LIN {X 0,Y 383.06,Z 302.767,A -85,B 0,C 180,E1 -12122.697,E2 -12122.697} C_VEL
LIN {X 0,Y 383.055,Z 302.766,A -85,B 0,C 180,E1 -12125.039,E2 -12125.039} C_VEL
LIN {X 0,Y 383.008,Z 302.777,A -85,B 0,C 180,E1 -12128.468,E2 -12128.468} C_VEL
LIN {X 0,Y 383.096,Z 302.761,A -85,B 0,C 180,E1 -12131.827,E2 -12131.827} C_VEL
LIN {X 0,Y 383.112,Z 302.76,A -85,B 0,C 180,E1 -12135.117,E2 -12135.117} C_VEL
LIN {X 0,Y 383.099,Z 302.764,A -85,B 0,C 180,E1 -12138.357,E2 -12138.357} C_VEL
LIN {X 0,Y 383.287,Z 302.941,A -85,B 0,C 180,E1 -12142.164,E2 -12142.164} C_VEL
LIN {X 0,Y 384.877,Z 312.371,A -85,B 0,C 180,E1 -12144.497,E2 -12144.497} C_VEL
LIN {X 0,Y 384.952,Z 313.789,A -85,B 0,C 180,E1 -12144.835,E2 -12144.835} C_VEL
LIN {X 0,Y 389.451,Z 337.201,A -85,B 0,C 180,E1 -12145.495,E2 -12145.495} C_VEL
LIN {X 0,Y 388.112,Z 421.744,A -85,B 0,C 180,E1 -12147.079,E2 -12147.079} C_VEL
LIN {X 0,Y 387.644,Z 434.738,A -85,B 0,C 180,E1 -12147.531,E2 -12147.531} C_VEL
LIN {X 0,Y 387.184,Z 447.368,A -85,B 0,C 180,E1 -12148.187,E2 -12148.187} C_VEL
LIN {X 0,Y 386.537,Z 458.426,A -85,B 0,C 180,E1 -12148.957,E2 -12148.957} C_VEL
LIN {X 0,Y 385.704,Z 470.032,A -85,B 0,C 180,E1 -12149.998,E2 -12149.998} C_VEL
LIN {X 0,Y 384.812,Z 480.494,A -85,B 0,C 180,E1 -12151.176,E2 -12151.176} C_VEL
LIN {X 0,Y 384.141,Z 489.023,A -85,B 0,C 180,E1 -12152.358,E2 -12152.358} C_VEL
LIN {X 0,Y 383.427,Z 496.909,A -85,B 0,C 180,E1 -12153.677,E2 -12153.677} C_VEL
LIN {X 0,Y 382.792,Z 504.598,A -85,B 0,C 180,E1 -12155.265,E2 -12155.265} C_VEL
LIN {X 0,Y 382.412,Z 511.451,A -85,B 0,C 180,E1 -12157.062,E2 -12157.062} C_VEL
LIN {X 0,Y 382.07,Z 515.669,A -85,B 0,C 180,E1 -12158.46,E2 -12158.46} C_VEL
LIN {X 0,Y 381.795,Z 519.452,A -85,B 0,C 180,E1 -12160.07,E2 -12160.07} C_VEL
LIN {X 0,Y 381.626,Z 522.196,A -85,B 0,C 180,E1 -12161.686,E2 -12161.686} C_VEL
LIN {X 0,Y 381.565,Z 523.488,A -85,B 0,C 180,E1 -12162.768,E2 -12162.768} C_VEL
LIN {X 0,Y 381.483,Z 524.406,A -85,B 0,C 180,E1 -12163.955,E2 -12163.955} C_VEL
LIN {X 0,Y 380.776,Z 524.798,A -85,B 0,C 180,E1 -12164.837,E2 -12164.837} C_VEL
LIN {X 0,Y 377.938,Z 524.939,A -85,B 0,C 180,E1 -12166.275,E2 -12166.275} C_VEL
LIN {X 0,Y 375.599,Z 524.604,A -85,B 0,C 180,E1 -12167.433,E2 -12167.433} C_VEL
LIN {X 0,Y 374.64,Z 523.917,A -85,B 0,C 180,E1 -12168.321,E2 -12168.321} C_VEL
LIN {X 0,Y 374.584,Z 523.586,A -85,B 0,C 180,E1 -12168.619,E2 -12168.619} C_VEL
LIN {X 0,Y 374.869,Z 521.239,A -85,B 0,C 180,E1 -12170.382,E2 -12170.382} C_VEL
LIN {X 0,Y 375.204,Z 518.078,A -85,B 0,C 180,E1 -12171.999,E2 -12171.999} C_VEL
LIN {X 0,Y 375.731,Z 513.289,A -85,B 0,C 180,E1 -12173.813,E2 -12173.813} C_VEL
LIN {X 0,Y 376.416,Z 507.759,A -85,B 0,C 180,E1 -12175.429,E2 -12175.429} C_VEL
LIN {X 0,Y 377.35,Z 500.326,A -85,B 0,C 180,E1 -12177.147,E2 -12177.147} C_VEL
LIN {X 0,Y 378.264,Z 492.622,A -85,B 0,C 180,E1 -12178.58,E2 -12178.58} C_VEL
LIN {X 0,Y 379.408,Z 483.177,A -85,B 0,C 180,E1 -12180.007,E2 -12180.007} C_VEL
LIN {X 0,Y 380.528,Z 472.847,A -85,B 0,C 180,E1 -12181.265,E2 -12181.265} C_VEL
LIN {X 0,Y 381.589,Z 462.332,A -85,B 0,C 180,E1 -12182.282,E2 -12182.282} C_VEL
LIN {X 0,Y 382.549,Z 450.16,A -85,B 0,C 180,E1 -12183.207,E2 -12183.207} C_VEL
LIN {X 0,Y 383.376,Z 437.639,A -85,B 0,C 180,E1 -12183.914,E2 -12183.914} C_VEL
LIN {X 0,Y 383.918,Z 424.605,A -85,B 0,C 180,E1 -12184.414,E2 -12184.414} C_VEL
LIN {X 0,Y 384.424,Z 405.525,A -85,B 0,C 180,E1 -12184.824,E2 -12184.824} C_VEL
LIN {X 0,Y 385.538,Z 338.341,A -85,B 0,C 180,E1 -12186.11,E2 -12186.11} C_VEL
LIN {X 0,Y 381.903,Z 323.107,A -85,B 0,C 180,E1 -12186.677,E2 -12186.677} C_VEL
LIN {X 0,Y 378.283,Z 314.275,A -85,B 0,C 180,E1 -12187.135,E2 -12187.135} C_VEL
LIN {X 0,Y 375.924,Z 303.662,A -85,B 0,C 180,E1 -12189.991,E2 -12189.991} C_VEL
LIN {X 0,Y 375.914,Z 303.66,A -85,B 0,C 180,E1 -12193.765,E2 -12193.765} C_VEL
LIN {X 0,Y 375.922,Z 303.652,A -85,B 0,C 180,E1 -12196.809,E2 -12196.809} C_VEL
LIN {X 0,Y 375.921,Z 303.658,A -85,B 0,C 180,E1 -12200.533,E2 -12200.533} C_VEL
LIN {X 0,Y 375.945,Z 303.646,A -85,B 0,C 180,E1 -12203.496,E2 -12203.496} C_VEL
LIN {X 0,Y 375.946,Z 303.65,A -85,B 0,C 180,E1 -12205.887,E2 -12205.887} C_VEL
LIN {X 0,Y 375.949,Z 303.655,A -85,B 0,C 180,E1 -12209.686,E2 -12209.686} C_VEL
LIN {X 0,Y 375.921,Z 303.656,A -85,B 0,C 180,E1 -12212.136,E2 -12212.136} C_VEL
LIN {X 0,Y 375.958,Z 303.649,A -85,B 0,C 180,E1 -12215.716,E2 -12215.716} C_VEL
LIN {X 0,Y 375.984,Z 303.642,A -85,B 0,C 180,E1 -12219.197,E2 -12219.197} C_VEL
LIN {X 0,Y 376.036,Z 303.637,A -85,B 0,C 180,E1 -12222.601,E2 -12222.601} C_VEL
LIN {X 0,Y 376.075,Z 303.638,A -85,B 0,C 180,E1 -12226.342,E2 -12226.342} C_VEL
LIN {X 0,Y 376.107,Z 303.639,A -85,B 0,C 180,E1 -12230.318,E2 -12230.318} C_VEL
LIN {X 0,Y 376.198,Z 303.613,A -85,B 0,C 180,E1 -12233.564,E2 -12233.564} C_VEL
LIN {X 0,Y 376.337,Z 303.598,A -85,B 0,C 180,E1 -12237.86,E2 -12237.86} C_VEL
LIN {X 0,Y 376.474,Z 303.585,A -85,B 0,C 180,E1 -12240,E2 -12240} C_VEL
LIN {X 0,Y 376.17,Z 303.614,A -85,B 0,C 180,E1 -12243.213,E2 -12243.213} C_VEL
LIN {X 0,Y 376.231,Z 303.62,A -85,B 0,C 180,E1 -12246.435,E2 -12246.435} C_VEL
LIN {X 0,Y 376.192,Z 303.615,A -85,B 0,C 180,E1 -12248.596,E2 -12248.596} C_VEL
LIN {X 0,Y 376.037,Z 303.64,A -85,B 0,C 180,E1 -12251.864,E2 -12251.864} C_VEL
LIN {X 0,Y 376.045,Z 303.642,A -85,B 0,C 180,E1 -12255.168,E2 -12255.168} C_VEL
LIN {X 0,Y 376.011,Z 303.64,A -85,B 0,C 180,E1 -12258.527,E2 -12258.527} C_VEL
LIN {X 0,Y 375.951,Z 303.652,A -85,B 0,C 180,E1 -12261.955,E2 -12261.955} C_VEL
LIN {X 0,Y 375.995,Z 303.65,A -85,B 0,C 180,E1 -12265.462,E2 -12265.462} C_VEL
LIN {X 0,Y 375.966,Z 303.649,A -85,B 0,C 180,E1 -12269.08,E2 -12269.08} C_VEL
LIN {X 0,Y 375.948,Z 303.65,A -85,B 0,C 180,E1 -12272.829,E2 -12272.829} C_VEL
LIN {X 0,Y 375.948,Z 303.654,A -85,B 0,C 180,E1 -12275.417,E2 -12275.417} C_VEL
LIN {X 0,Y 375.968,Z 303.652,A -85,B 0,C 180,E1 -12278.273,E2 -12278.273} C_VEL
LIN {X 0,Y 375.953,Z 303.655,A -85,B 0,C 180,E1 -12281.607,E2 -12281.607} C_VEL
LIN {X 0,Y 375.972,Z 303.643,A -85,B 0,C 180,E1 -12285.262,E2 -12285.262} C_VEL
LIN {X 0,Y 375.982,Z 303.65,A -85,B 0,C 180,E1 -12288.391,E2 -12288.391} C_VEL
LIN {X 0,Y 375.962,Z 303.658,A -85,B 0,C 180,E1 -12291.914,E2 -12291.914} C_VEL
LIN {X 0,Y 375.975,Z 303.656,A -85,B 0,C 180,E1 -12295.334,E2 -12295.334} C_VEL
LIN {X 0,Y 375.953,Z 303.651,A -85,B 0,C 180,E1 -12298.44,E2 -12298.44} C_VEL
LIN {X 0,Y 375.963,Z 303.774,A -85,B 0,C 180,E1 -12299.481,E2 -12299.481} C_VEL
LIN {X 0,Y 378.342,Z 313.599,A -85,B 0,C 180,E1 -12302.03,E2 -12302.03} C_VEL
LIN {X 0,Y 380.138,Z 322.611,A -85,B 0,C 180,E1 -12304.251,E2 -12304.251} C_VEL
LIN {X 0,Y 380.37,Z 326.084,A -85,B 0,C 180,E1 -12305.056,E2 -12305.056} C_VEL
LIN {X 0,Y 379.02,Z 339.738,A -85,B 0,C 180,E1 -12307.992,E2 -12307.992} C_VEL
LIN {X 0,Y 383.174,Z 360.734,A -85,B 0,C 180,E1 -12308.716,E2 -12308.716} C_VEL
LIN {X 0,Y 385.058,Z 374.292,A -85,B 0,C 180,E1 -12309.118,E2 -12309.118} C_VEL
LIN {X 0,Y 383.66,Z 448.299,A -85,B 0,C 180,E1 -12310.547,E2 -12310.547} C_VEL
LIN {X 0,Y 382.984,Z 462.066,A -85,B 0,C 180,E1 -12311.027,E2 -12311.027} C_VEL
LIN {X 0,Y 382.088,Z 474.003,A -85,B 0,C 180,E1 -12311.642,E2 -12311.642} C_VEL
LIN {X 0,Y 381.049,Z 485.315,A -85,B 0,C 180,E1 -12312.423,E2 -12312.423} C_VEL
LIN {X 0,Y 379.899,Z 496.976,A -85,B 0,C 180,E1 -12313.477,E2 -12313.477} C_VEL
LIN {X 0,Y 378.675,Z 507.472,A -85,B 0,C 180,E1 -12314.666,E2 -12314.666} C_VEL
LIN {X 0,Y 377.746,Z 516.955,A -85,B 0,C 180,E1 -12316.005,E2 -12316.005} C_VEL
LIN {X 0,Y 376.624,Z 526.113,A -85,B 0,C 180,E1 -12317.61,E2 -12317.61} C_VEL
LIN {X 0,Y 375.732,Z 533.511,A -85,B 0,C 180,E1 -12319.221,E2 -12319.221} C_VEL
LIN {X 0,Y 375.192,Z 539.471,A -85,B 0,C 180,E1 -12320.84,E2 -12320.84} C_VEL
LIN {X 0,Y 374.802,Z 544.195,A -85,B 0,C 180,E1 -12322.459,E2 -12322.459} C_VEL
LIN {X 0,Y 374.589,Z 547.514,A -85,B 0,C 180,E1 -12323.925,E2 -12323.925} C_VEL
LIN {X 0,Y 374.551,Z 550.446,A -85,B 0,C 180,E1 -12325.697,E2 -12325.697} C_VEL
LIN {X 0,Y 374.463,Z 551.691,A -85,B 0,C 180,E1 -12326.774,E2 -12326.774} C_VEL
LIN {X 0,Y 374.496,Z 552.514,A -85,B 0,C 180,E1 -12327.851,E2 -12327.851} C_VEL
LIN {X 0,Y 374.555,Z 552.921,A -85,B 0,C 180,E1 -12328.926,E2 -12328.926} C_VEL
LIN {X 0,Y 374.589,Z 552.942,A -85,B 0,C 180,E1 -12330.002,E2 -12330.002} C_VEL
LIN {X 0,Y 374.586,Z 552.575,A -85,B 0,C 180,E1 -12331.077,E2 -12331.077} C_VEL
LIN {X 0,Y 374.525,Z 551.793,A -85,B 0,C 180,E1 -12332.152,E2 -12332.152} C_VEL
LIN {X 0,Y 374.56,Z 548.949,A -85,B 0,C 180,E1 -12334.306,E2 -12334.306} C_VEL
LIN {X 0,Y 374.588,Z 545.319,A -85,B 0,C 180,E1 -12336.073,E2 -12336.073} C_VEL
LIN {X 0,Y 374.771,Z 541.297,A -85,B 0,C 180,E1 -12337.544,E2 -12337.544} C_VEL
LIN {X 0,Y 375.078,Z 535.718,A -85,B 0,C 180,E1 -12339.166,E2 -12339.166} C_VEL
LIN {X 0,Y 375.526,Z 528.739,A -85,B 0,C 180,E1 -12340.788,E2 -12340.788} C_VEL
LIN {X 0,Y 376.325,Z 519.99,A -85,B 0,C 180,E1 -12342.403,E2 -12342.403} C_VEL
LIN {X 0,Y 377.094,Z 511.006,A -85,B 0,C 180,E1 -12343.748,E2 -12343.748} C_VEL
LIN {X 0,Y 377.801,Z 501.585,A -85,B 0,C 180,E1 -12344.905,E2 -12344.905} C_VEL
LIN {X 0,Y 378.647,Z 490.228,A -85,B 0,C 180,E1 -12346.029,E2 -12346.029} C_VEL
LIN {X 0,Y 379.538,Z 477.995,A -85,B 0,C 180,E1 -12346.958,E2 -12346.958} C_VEL
LIN {X 0,Y 380.371,Z 465.206,A -85,B 0,C 180,E1 -12347.682,E2 -12347.682} C_VEL
LIN {X 0,Y 381.01,Z 452.494,A -85,B 0,C 180,E1 -12348.172,E2 -12348.172} C_VEL
LIN {X 0,Y 381.368,Z 434.485,A -85,B 0,C 180,E1 -12348.572,E2 -12348.572} C_VEL
LIN {X 0,Y 382.075,Z 371.258,A -85,B 0,C 180,E1 -12349.767,E2 -12349.767} C_VEL
LIN {X 0,Y 377.67,Z 340.16,A -85,B 0,C 180,E1 -12350.591,E2 -12350.591} C_VEL
LIN {X 0,Y 378.973,Z 323.714,A -85,B 0,C 180,E1 -12354.08,E2 -12354.08} C_VEL
LIN {X 0,Y 379.156,Z 319.824,A -85,B 0,C 180,E1 -12354.918,E2 -12354.918} C_VEL
LIN {X 0,Y 376.815,Z 307.387,A -85,B 0,C 180,E1 -12357.794,E2 -12357.794} C_VEL
LIN {X 0,Y 376.048,Z 303.644,A -85,B 0,C 180,E1 -12358.687,E2 -12358.687} C_VEL
LIN {X 0,Y 375.955,Z 303.652,A -85,B 0,C 180,E1 -12362.731,E2 -12362.731} C_VEL
LIN {X 0,Y 375.963,Z 303.649,A -85,B 0,C 180,E1 -12365.416,E2 -12365.416} C_VEL
LIN {X 0,Y 375.978,Z 303.653,A -85,B 0,C 180,E1 -12368.271,E2 -12368.271} C_VEL
LIN {X 0,Y 375.94,Z 303.652,A -85,B 0,C 180,E1 -12371.601,E2 -12371.601} C_VEL
LIN {X 0,Y 375.933,Z 303.654,A -85,B 0,C 180,E1 -12375.269,E2 -12375.269} C_VEL
LIN {X 0,Y 375.941,Z 303.655,A -85,B 0,C 180,E1 -12378.4,E2 -12378.4} C_VEL
LIN {X 0,Y 375.979,Z 303.647,A -85,B 0,C 180,E1 -12381.73,E2 -12381.73} C_VEL
LIN {X 0,Y 375.985,Z 303.649,A -85,B 0,C 180,E1 -12385.333,E2 -12385.333} C_VEL
LIN {X 0,Y 375.963,Z 303.65,A -85,B 0,C 180,E1 -12388.438,E2 -12388.438} C_VEL
LIN {X 0,Y 375.99,Z 303.646,A -85,B 0,C 180,E1 -12392.141,E2 -12392.141} C_VEL
LIN {X 0,Y 376.012,Z 303.643,A -85,B 0,C 180,E1 -12394.539,E2 -12394.539} C_VEL
LIN {X 0,Y 375.964,Z 303.65,A -85,B 0,C 180,E1 -12398.045,E2 -12398.045} C_VEL
LIN {X 0,Y 376.009,Z 303.651,A -85,B 0,C 180,E1 -12401.473,E2 -12401.473} C_VEL
LIN {X 0,Y 376.065,Z 303.637,A -85,B 0,C 180,E1 -12404.833,E2 -12404.833} C_VEL
LIN {X 0,Y 376.055,Z 303.64,A -85,B 0,C 180,E1 -12408.137,E2 -12408.137} C_VEL
LIN {X 0,Y 376.194,Z 303.626,A -85,B 0,C 180,E1 -12411.953,E2 -12411.953} C_VEL
LIN {X 0,Y 376.161,Z 303.625,A -85,B 0,C 180,E1 -12414.64,E2 -12414.64} C_VEL
LIN {X 0,Y 376.357,Z 303.605,A -85,B 0,C 180,E1 -12417.859,E2 -12417.859} C_VEL
LIN {X 0,Y 376.491,Z 303.589,A -85,B 0,C 180,E1 -12420,E2 -12420} C_VEL
LIN {X 0,Y 376.187,Z 303.621,A -85,B 0,C 180,E1 -12423.213,E2 -12423.213} C_VEL
LIN {X 0,Y 376.219,Z 303.621,A -85,B 0,C 180,E1 -12426.593,E2 -12426.593} C_VEL
LIN {X 0,Y 376.119,Z 303.63,A -85,B 0,C 180,E1 -12429.681,E2 -12429.681} C_VEL
LIN {X 0,Y 376.095,Z 303.633,A -85,B 0,C 180,E1 -12433.657,E2 -12433.657} C_VEL
LIN {X 0,Y 376.038,Z 303.64,A -85,B 0,C 180,E1 -12437.399,E2 -12437.399} C_VEL
LIN {X 0,Y 375.984,Z 303.653,A -85,B 0,C 180,E1 -12440.832,E2 -12440.832} C_VEL
LIN {X 0,Y 375.995,Z 303.646,A -85,B 0,C 180,E1 -12444.281,E2 -12444.281} C_VEL
LIN {X 0,Y 376.025,Z 303.645,A -85,B 0,C 180,E1 -12446.651,E2 -12446.651} C_VEL
LIN {X 0,Y 375.97,Z 303.648,A -85,B 0,C 180,E1 -12450.312,E2 -12450.312} C_VEL
LIN {X 0,Y 375.965,Z 303.649,A -85,B 0,C 180,E1 -12454.111,E2 -12454.111} C_VEL
LIN {X 0,Y 375.958,Z 303.651,A -85,B 0,C 180,E1 -12456.74,E2 -12456.74} C_VEL
LIN {X 0,Y 375.993,Z 303.647,A -85,B 0,C 180,E1 -12459.97,E2 -12459.97} C_VEL
LIN {X 0,Y 375.934,Z 303.657,A -85,B 0,C 180,E1 -12463.765,E2 -12463.765} C_VEL
LIN {X 0,Y 375.938,Z 303.652,A -85,B 0,C 180,E1 -12466.81,E2 -12466.81} C_VEL
LIN {X 0,Y 375.965,Z 303.649,A -85,B 0,C 180,E1 -12470.536,E2 -12470.536} C_VEL
LIN {X 0,Y 375.967,Z 303.651,A -85,B 0,C 180,E1 -12473.495,E2 -12473.495} C_VEL
LIN {X 0,Y 375.964,Z 303.656,A -85,B 0,C 180,E1 -12475.888,E2 -12475.888} C_VEL
LIN {X 0,Y 375.968,Z 303.651,A -85,B 0,C 180,E1 -12479.686,E2 -12479.686} C_VEL
LIN {X 0,Y 376.023,Z 303.642,A -85,B 0,C 180,E1 -12483.347,E2 -12483.347} C_VEL
LIN {X 0,Y 376.001,Z 303.646,A -85,B 0,C 180,E1 -12486.887,E2 -12486.887} C_VEL
LIN {X 0,Y 376.014,Z 303.649,A -85,B 0,C 180,E1 -12490.339,E2 -12490.339} C_VEL
LIN {X 0,Y 376.031,Z 303.641,A -85,B 0,C 180,E1 -12493.718,E2 -12493.718} C_VEL
LIN {X 0,Y 376.105,Z 303.634,A -85,B 0,C 180,E1 -12497.041,E2 -12497.041} C_VEL
LIN {X 0,Y 376.115,Z 303.633,A -85,B 0,C 180,E1 -12500.317,E2 -12500.317} C_VEL
LIN {X 0,Y 376.211,Z 303.756,A -85,B 0,C 180,E1 -12501.927,E2 -12501.927} C_VEL
LIN {X 0,Y 377.946,Z 313.948,A -85,B 0,C 180,E1 -12504.496,E2 -12504.496} C_VEL
LIN {X 0,Y 382.58,Z 337.48,A -85,B 0,C 180,E1 -12505.193,E2 -12505.193} C_VEL
LIN {X 0,Y 381.288,Z 421.788,A -85,B 0,C 180,E1 -12506.801,E2 -12506.801} C_VEL
LIN {X 0,Y 380.809,Z 434.724,A -85,B 0,C 180,E1 -12507.255,E2 -12507.255} C_VEL
LIN {X 0,Y 380.287,Z 447.792,A -85,B 0,C 180,E1 -12507.943,E2 -12507.943} C_VEL
LIN {X 0,Y 379.523,Z 460.257,A -85,B 0,C 180,E1 -12508.848,E2 -12508.848} C_VEL
LIN {X 0,Y 378.7,Z 471.157,A -85,B 0,C 180,E1 -12509.866,E2 -12509.866} C_VEL
LIN {X 0,Y 377.781,Z 481.471,A -85,B 0,C 180,E1 -12511.064,E2 -12511.064} C_VEL
LIN {X 0,Y 377.043,Z 490.693,A -85,B 0,C 180,E1 -12512.402,E2 -12512.402} C_VEL
LIN {X 0,Y 376.198,Z 499.683,A -85,B 0,C 180,E1 -12514.016,E2 -12514.016} C_VEL
LIN {X 0,Y 375.595,Z 506.918,A -85,B 0,C 180,E1 -12515.636,E2 -12515.636} C_VEL
LIN {X 0,Y 375.329,Z 512.018,A -85,B 0,C 180,E1 -12517.06,E2 -12517.06} C_VEL
LIN {X 0,Y 374.951,Z 516.536,A -85,B 0,C 180,E1 -12518.622,E2 -12518.622} C_VEL
LIN {X 0,Y 374.689,Z 520.169,A -85,B 0,C 180,E1 -12520.263,E2 -12520.263} C_VEL
LIN {X 0,Y 374.527,Z 522.771,A -85,B 0,C 180,E1 -12521.911,E2 -12521.911} C_VEL
LIN {X 0,Y 374.469,Z 523.984,A -85,B 0,C 180,E1 -12523.014,E2 -12523.014} C_VEL
LIN {X 0,Y 374.391,Z 524.74,A -85,B 0,C 180,E1 -12524.123,E2 -12524.123} C_VEL
LIN {X 0,Y 374.37,Z 525.094,A -85,B 0,C 180,E1 -12525.236,E2 -12525.236} C_VEL
LIN {X 0,Y 374.419,Z 524.881,A -85,B 0,C 180,E1 -12526.806,E2 -12526.806} C_VEL
LIN {X 0,Y 374.584,Z 523.586,A -85,B 0,C 180,E1 -12528.619,E2 -12528.619} C_VEL
LIN {X 0,Y 374.025,Z 522.607,A -85,B 0,C 180,E1 -12529.504,E2 -12529.504} C_VEL
LIN {X 0,Y 371.432,Z 520.566,A -85,B 0,C 180,E1 -12530.943,E2 -12530.943} C_VEL
LIN {X 0,Y 369.294,Z 518.495,A -85,B 0,C 180,E1 -12532.088,E2 -12532.088} C_VEL
LIN {X 0,Y 368.495,Z 516.557,A -85,B 0,C 180,E1 -12532.95,E2 -12532.95} C_VEL
LIN {X 0,Y 368.494,Z 515.813,A -85,B 0,C 180,E1 -12533.236,E2 -12533.236} C_VEL
LIN {X 0,Y 369.194,Z 510.33,A -85,B 0,C 180,E1 -12535.057,E2 -12535.057} C_VEL
LIN {X 0,Y 370.042,Z 503.558,A -85,B 0,C 180,E1 -12536.793,E2 -12536.793} C_VEL
LIN {X 0,Y 371.218,Z 494.867,A -85,B 0,C 180,E1 -12538.555,E2 -12538.555} C_VEL
LIN {X 0,Y 372.402,Z 485.874,A -85,B 0,C 180,E1 -12540.008,E2 -12540.008} C_VEL
LIN {X 0,Y 373.495,Z 475.851,A -85,B 0,C 180,E1 -12541.318,E2 -12541.318} C_VEL
LIN {X 0,Y 374.701,Z 465.159,A -85,B 0,C 180,E1 -12542.432,E2 -12542.432} C_VEL
LIN {X 0,Y 375.757,Z 453.329,A -85,B 0,C 180,E1 -12543.405,E2 -12543.405} C_VEL
LIN {X 0,Y 376.573,Z 441.882,A -85,B 0,C 180,E1 -12544.117,E2 -12544.117} C_VEL
LIN {X 0,Y 377.262,Z 429.042,A -85,B 0,C 180,E1 -12544.69,E2 -12544.69} C_VEL
LIN {X 0,Y 377.683,Z 417.058,A -85,B 0,C 180,E1 -12545.028,E2 -12545.028} C_VEL
LIN {X 0,Y 379.109,Z 339.423,A -85,B 0,C 180,E1 -12546.54,E2 -12546.54} C_VEL
LIN {X 0,Y 375.745,Z 325.617,A -85,B 0,C 180,E1 -12547.075,E2 -12547.075} C_VEL
LIN {X 0,Y 371.138,Z 314.54,A -85,B 0,C 180,E1 -12547.677,E2 -12547.677} C_VEL
LIN {X 0,Y 368.862,Z 304.537,A -85,B 0,C 180,E1 -12550.463,E2 -12550.463} C_VEL
LIN {X 0,Y 368.868,Z 304.539,A -85,B 0,C 180,E1 -12553.614,E2 -12553.614} C_VEL
LIN {X 0,Y 368.873,Z 304.529,A -85,B 0,C 180,E1 -12556.694,E2 -12556.694} C_VEL
LIN {X 0,Y 368.872,Z 304.541,A -85,B 0,C 180,E1 -12559.647,E2 -12559.647} C_VEL
LIN {X 0,Y 368.883,Z 304.531,A -85,B 0,C 180,E1 -12563.144,E2 -12563.144} C_VEL
LIN {X 0,Y 368.883,Z 304.535,A -85,B 0,C 180,E1 -12566.461,E2 -12566.461} C_VEL
LIN {X 0,Y 368.899,Z 304.528,A -85,B 0,C 180,E1 -12569.044,E2 -12569.044} C_VEL
LIN {X 0,Y 368.903,Z 304.53,A -85,B 0,C 180,E1 -12571.558,E2 -12571.558} C_VEL
LIN {X 0,Y 368.912,Z 304.526,A -85,B 0,C 180,E1 -12575.222,E2 -12575.222} C_VEL
LIN {X 0,Y 368.906,Z 304.523,A -85,B 0,C 180,E1 -12578.98,E2 -12578.98} C_VEL
LIN {X 0,Y 368.977,Z 304.519,A -85,B 0,C 180,E1 -12582.257,E2 -12582.257} C_VEL
LIN {X 0,Y 369.023,Z 304.518,A -85,B 0,C 180,E1 -12586.228,E2 -12586.228} C_VEL
LIN {X 0,Y 369.055,Z 304.514,A -85,B 0,C 180,E1 -12590.132,E2 -12590.132} C_VEL
LIN {X 0,Y 369.158,Z 304.489,A -85,B 0,C 180,E1 -12593.441,E2 -12593.441} C_VEL
LIN {X 0,Y 369.302,Z 304.474,A -85,B 0,C 180,E1 -12597.819,E2 -12597.819} C_VEL
LIN {X 0,Y 369.444,Z 304.461,A -85,B 0,C 180,E1 -12600,E2 -12600} C_VEL
LIN {X 0,Y 369.302,Z 304.48,A -85,B 0,C 180,E1 -12602.181,E2 -12602.181} C_VEL
LIN {X 0,Y 369.193,Z 304.497,A -85,B 0,C 180,E1 -12606.559,E2 -12606.559} C_VEL
LIN {X 0,Y 369.124,Z 304.496,A -85,B 0,C 180,E1 -12608.761,E2 -12608.761} C_VEL
LIN {X 0,Y 368.992,Z 304.518,A -85,B 0,C 180,E1 -12612.094,E2 -12612.094} C_VEL
LIN {X 0,Y 368.984,Z 304.521,A -85,B 0,C 180,E1 -12615.466,E2 -12615.466} C_VEL
LIN {X 0,Y 368.969,Z 304.516,A -85,B 0,C 180,E1 -12618.894,E2 -12618.894} C_VEL
LIN {X 0,Y 368.92,Z 304.528,A -85,B 0,C 180,E1 -12622.396,E2 -12622.396} C_VEL
LIN {X 0,Y 368.988,Z 304.52,A -85,B 0,C 180,E1 -12625.981,E2 -12625.981} C_VEL
LIN {X 0,Y 368.957,Z 304.519,A -85,B 0,C 180,E1 -12628.815,E2 -12628.815} C_VEL
LIN {X 0,Y 368.9,Z 304.525,A -85,B 0,C 180,E1 -12632.238,E2 -12632.238} C_VEL
LIN {X 0,Y 368.919,Z 304.533,A -85,B 0,C 180,E1 -12635.003,E2 -12635.003} C_VEL
LIN {X 0,Y 368.904,Z 304.532,A -85,B 0,C 180,E1 -12638.643,E2 -12638.643} C_VEL
LIN {X 0,Y 368.902,Z 304.531,A -85,B 0,C 180,E1 -12641.82,E2 -12641.82} C_VEL
LIN {X 0,Y 368.947,Z 304.519,A -85,B 0,C 180,E1 -12645.189,E2 -12645.189} C_VEL
LIN {X 0,Y 368.939,Z 304.529,A -85,B 0,C 180,E1 -12648.188,E2 -12648.188} C_VEL
LIN {X 0,Y 368.907,Z 304.531,A -85,B 0,C 180,E1 -12651.361,E2 -12651.361} C_VEL
LIN {X 0,Y 368.931,Z 304.532,A -85,B 0,C 180,E1 -12655.148,E2 -12655.148} C_VEL
LIN {X 0,Y 368.912,Z 304.617,A -85,B 0,C 180,E1 -12659.013,E2 -12659.013} C_VEL
LIN {X 0,Y 371.654,Z 316,A -85,B 0,C 180,E1 -12662.03,E2 -12662.03} C_VEL
LIN {X 0,Y 373.439,Z 325.27,A -85,B 0,C 180,E1 -12664.353,E2 -12664.353} C_VEL
LIN {X 0,Y 373.311,Z 329.368,A -85,B 0,C 180,E1 -12665.289,E2 -12665.289} C_VEL
LIN {X 0,Y 372.255,Z 339.389,A -85,B 0,C 180,E1 -12667.488,E2 -12667.488} C_VEL
LIN {X 0,Y 376.304,Z 359.631,A -85,B 0,C 180,E1 -12668.212,E2 -12668.212} C_VEL
LIN {X 0,Y 378.598,Z 374.173,A -85,B 0,C 180,E1 -12668.677,E2 -12668.677} C_VEL
LIN {X 0,Y 377.141,Z 447.747,A -85,B 0,C 180,E1 -12670.12,E2 -12670.12} C_VEL
LIN {X 0,Y 376.499,Z 460.975,A -85,B 0,C 180,E1 -12670.581,E2 -12670.581} C_VEL
LIN {X 0,Y 375.488,Z 473.687,A -85,B 0,C 180,E1 -12671.236,E2 -12671.236} C_VEL
LIN {X 0,Y 374.321,Z 485.813,A -85,B 0,C 180,E1 -12672.097,E2 -12672.097} C_VEL
LIN {X 0,Y 373.126,Z 497.323,A -85,B 0,C 180,E1 -12673.168,E2 -12673.168} C_VEL
LIN {X 0,Y 371.847,Z 507.715,A -85,B 0,C 180,E1 -12674.378,E2 -12674.378} C_VEL
LIN {X 0,Y 370.977,Z 515.952,A -85,B 0,C 180,E1 -12675.561,E2 -12675.561} C_VEL
LIN {X 0,Y 369.898,Z 524.814,A -85,B 0,C 180,E1 -12677.102,E2 -12677.102} C_VEL
LIN {X 0,Y 368.833,Z 532.387,A -85,B 0,C 180,E1 -12678.739,E2 -12678.739} C_VEL
LIN {X 0,Y 368.156,Z 539.411,A -85,B 0,C 180,E1 -12680.664,E2 -12680.664} C_VEL
LIN {X 0,Y 367.728,Z 544.087,A -85,B 0,C 180,E1 -12682.313,E2 -12682.313} C_VEL
LIN {X 0,Y 367.506,Z 547.638,A -85,B 0,C 180,E1 -12683.948,E2 -12683.948} C_VEL
LIN {X 0,Y 367.456,Z 550.258,A -85,B 0,C 180,E1 -12685.614,E2 -12685.614} C_VEL
LIN {X 0,Y 367.381,Z 551.484,A -85,B 0,C 180,E1 -12686.712,E2 -12686.712} C_VEL
LIN {X 0,Y 367.396,Z 552.273,A -85,B 0,C 180,E1 -12687.809,E2 -12687.809} C_VEL
LIN {X 0,Y 367.457,Z 552.664,A -85,B 0,C 180,E1 -12688.906,E2 -12688.906} C_VEL
LIN {X 0,Y 367.505,Z 552.669,A -85,B 0,C 180,E1 -12690.002,E2 -12690.002} C_VEL
LIN {X 0,Y 367.488,Z 552.283,A -85,B 0,C 180,E1 -12691.097,E2 -12691.097} C_VEL
LIN {X 0,Y 367.426,Z 551.467,A -85,B 0,C 180,E1 -12692.194,E2 -12692.194} C_VEL
LIN {X 0,Y 367.489,Z 548.587,A -85,B 0,C 180,E1 -12694.389,E2 -12694.389} C_VEL
LIN {X 0,Y 367.516,Z 545.199,A -85,B 0,C 180,E1 -12696.067,E2 -12696.067} C_VEL
LIN {X 0,Y 367.699,Z 540.854,A -85,B 0,C 180,E1 -12697.69,E2 -12697.69} C_VEL
LIN {X 0,Y 368.02,Z 535.23,A -85,B 0,C 180,E1 -12699.343,E2 -12699.343} C_VEL
LIN {X 0,Y 368.502,Z 528.19,A -85,B 0,C 180,E1 -12700.996,E2 -12700.996} C_VEL
LIN {X 0,Y 369.354,Z 519.36,A -85,B 0,C 180,E1 -12702.641,E2 -12702.641} C_VEL
LIN {X 0,Y 370.254,Z 509.311,A -85,B 0,C 180,E1 -12704.147,E2 -12704.147} C_VEL
LIN {X 0,Y 371.052,Z 499.039,A -85,B 0,C 180,E1 -12705.379,E2 -12705.379} C_VEL
LIN {X 0,Y 371.93,Z 487.628,A -85,B 0,C 180,E1 -12706.467,E2 -12706.467} C_VEL
LIN {X 0,Y 372.797,Z 475.79,A -85,B 0,C 180,E1 -12707.345,E2 -12707.345} C_VEL
LIN {X 0,Y 373.632,Z 462.812,A -85,B 0,C 180,E1 -12708.047,E2 -12708.047} C_VEL
LIN {X 0,Y 374.216,Z 450.051,A -85,B 0,C 180,E1 -12708.514,E2 -12708.514} C_VEL
LIN {X 0,Y 374.758,Z 421.996,A -85,B 0,C 180,E1 -12709.087,E2 -12709.087} C_VEL
LIN {X 0,Y 375.275,Z 372.109,A -85,B 0,C 180,E1 -12710.049,E2 -12710.049} C_VEL
LIN {X 0,Y 370.755,Z 339.901,A -85,B 0,C 180,E1 -12710.922,E2 -12710.922} C_VEL
LIN {X 0,Y 372.145,Z 323.117,A -85,B 0,C 180,E1 -12714.551,E2 -12714.551} C_VEL
LIN {X 0,Y 371.987,Z 319.75,A -85,B 0,C 180,E1 -12715.306,E2 -12715.306} C_VEL
LIN {X 0,Y 369.472,Z 306.704,A -85,B 0,C 180,E1 -12718.396,E2 -12718.396} C_VEL
LIN {X 0,Y 368.991,Z 304.521,A -85,B 0,C 180,E1 -12718.961,E2 -12718.961} C_VEL
LIN {X 0,Y 368.904,Z 304.535,A -85,B 0,C 180,E1 -12722.239,E2 -12722.239} C_VEL
LIN {X 0,Y 368.935,Z 304.525,A -85,B 0,C 180,E1 -12725.002,E2 -12725.002} C_VEL
LIN {X 0,Y 368.912,Z 304.532,A -85,B 0,C 180,E1 -12728.641,E2 -12728.641} C_VEL
LIN {X 0,Y 368.887,Z 304.532,A -85,B 0,C 180,E1 -12732.01,E2 -12732.01} C_VEL
LIN {X 0,Y 368.886,Z 304.532,A -85,B 0,C 180,E1 -12735.176,E2 -12735.176} C_VEL
LIN {X 0,Y 368.889,Z 304.532,A -85,B 0,C 180,E1 -12738.178,E2 -12738.178} C_VEL
LIN {X 0,Y 368.914,Z 304.529,A -85,B 0,C 180,E1 -12741.36,E2 -12741.36} C_VEL
LIN {X 0,Y 368.942,Z 304.529,A -85,B 0,C 180,E1 -12745.147,E2 -12745.147} C_VEL
LIN {X 0,Y 368.936,Z 304.531,A -85,B 0,C 180,E1 -12749.047,E2 -12749.047} C_VEL
LIN {X 0,Y 368.982,Z 304.521,A -85,B 0,C 180,E1 -12751.564,E2 -12751.564} C_VEL
LIN {X 0,Y 369.006,Z 304.516,A -85,B 0,C 180,E1 -12754.02,E2 -12754.02} C_VEL
LIN {X 0,Y 368.929,Z 304.53,A -85,B 0,C 180,E1 -12757.604,E2 -12757.604} C_VEL
LIN {X 0,Y 368.961,Z 304.524,A -85,B 0,C 180,E1 -12761.106,E2 -12761.106} C_VEL
LIN {X 0,Y 369.003,Z 304.516,A -85,B 0,C 180,E1 -12764.535,E2 -12764.535} C_VEL
LIN {X 0,Y 369.011,Z 304.52,A -85,B 0,C 180,E1 -12767.907,E2 -12767.907} C_VEL
LIN {X 0,Y 369.098,Z 304.505,A -85,B 0,C 180,E1 -12771.238,E2 -12771.238} C_VEL
LIN {X 0,Y 369.132,Z 304.501,A -85,B 0,C 180,E1 -12774.537,E2 -12774.537} C_VEL
LIN {X 0,Y 369.322,Z 304.481,A -85,B 0,C 180,E1 -12777.819,E2 -12777.819} C_VEL
LIN {X 0,Y 369.46,Z 304.465,A -85,B 0,C 180,E1 -12780,E2 -12780} C_VEL
LIN {X 0,Y 369.321,Z 304.484,A -85,B 0,C 180,E1 -12782.181,E2 -12782.181} C_VEL
LIN {X 0,Y 369.191,Z 304.497,A -85,B 0,C 180,E1 -12786.575,E2 -12786.575} C_VEL
LIN {X 0,Y 369.069,Z 304.509,A -85,B 0,C 180,E1 -12789.868,E2 -12789.868} C_VEL
LIN {X 0,Y 369.043,Z 304.511,A -85,B 0,C 180,E1 -12793.772,E2 -12793.772} C_VEL
LIN {X 0,Y 368.997,Z 304.517,A -85,B 0,C 180,E1 -12797.742,E2 -12797.742} C_VEL
LIN {X 0,Y 368.916,Z 304.529,A -85,B 0,C 180,E1 -12801.22,E2 -12801.22} C_VEL
LIN {X 0,Y 368.961,Z 304.527,A -85,B 0,C 180,E1 -12804.775,E2 -12804.775} C_VEL
LIN {X 0,Y 368.968,Z 304.525,A -85,B 0,C 180,E1 -12807.203,E2 -12807.203} C_VEL
LIN {X 0,Y 368.935,Z 304.53,A -85,B 0,C 180,E1 -12810.953,E2 -12810.953} C_VEL
LIN {X 0,Y 368.934,Z 304.529,A -85,B 0,C 180,E1 -12815.001,E2 -12815.001} C_VEL
LIN {X 0,Y 368.913,Z 304.528,A -85,B 0,C 180,E1 -12818.639,E2 -12818.639} C_VEL
LIN {X 0,Y 368.886,Z 304.532,A -85,B 0,C 180,E1 -12822.009,E2 -12822.009} C_VEL
LIN {X 0,Y 368.884,Z 304.533,A -85,B 0,C 180,E1 -12825.175,E2 -12825.175} C_VEL
LIN {X 0,Y 368.887,Z 304.532,A -85,B 0,C 180,E1 -12828.177,E2 -12828.177} C_VEL
LIN {X 0,Y 368.91,Z 304.53,A -85,B 0,C 180,E1 -12831.359,E2 -12831.359} C_VEL
LIN {X 0,Y 368.94,Z 304.524,A -85,B 0,C 180,E1 -12835.145,E2 -12835.145} C_VEL
LIN {X 0,Y 368.933,Z 304.525,A -85,B 0,C 180,E1 -12839.045,E2 -12839.045} C_VEL
LIN {X 0,Y 368.967,Z 304.522,A -85,B 0,C 180,E1 -12842.795,E2 -12842.795} C_VEL
LIN {X 0,Y 368.948,Z 304.528,A -85,B 0,C 180,E1 -12846.112,E2 -12846.112} C_VEL
LIN {X 0,Y 368.948,Z 304.525,A -85,B 0,C 180,E1 -12849.946,E2 -12849.946} C_VEL
LIN {X 0,Y 368.978,Z 304.519,A -85,B 0,C 180,E1 -12853.397,E2 -12853.397} C_VEL
LIN {X 0,Y 369.06,Z 304.514,A -85,B 0,C 180,E1 -12856.789,E2 -12856.789} C_VEL
LIN {X 0,Y 369.065,Z 304.509,A -85,B 0,C 180,E1 -12860.13,E2 -12860.13} C_VEL
LIN {X 0,Y 369.121,Z 304.516,A -85,B 0,C 180,E1 -12861.667,E2 -12861.667} C_VEL
LIN {X 0,Y 370.872,Z 314.396,A -85,B 0,C 180,E1 -12864.186,E2 -12864.186} C_VEL
LIN {X 0,Y 374.752,Z 332.838,A -85,B 0,C 180,E1 -12864.741,E2 -12864.741} C_VEL
LIN {X 0,Y 375.842,Z 339.479,A -85,B 0,C 180,E1 -12864.925,E2 -12864.925} C_VEL
LIN {X 0,Y 374.437,Z 422.389,A -85,B 0,C 180,E1 -12866.535,E2 -12866.535} C_VEL
LIN {X 0,Y 373.928,Z 435.354,A -85,B 0,C 180,E1 -12867.002,E2 -12867.002} C_VEL
LIN {X 0,Y 373.388,Z 448.366,A -85,B 0,C 180,E1 -12867.706,E2 -12867.706} C_VEL
LIN {X 0,Y 372.588,Z 460.898,A -85,B 0,C 180,E1 -12868.64,E2 -12868.64} C_VEL
LIN {X 0,Y 371.695,Z 472.23,A -85,B 0,C 180,E1 -12869.728,E2 -12869.728} C_VEL
LIN {X 0,Y 370.777,Z 482.363,A -85,B 0,C 180,E1 -12870.949,E2 -12870.949} C_VEL
LIN {X 0,Y 369.909,Z 492.295,A -85,B 0,C 180,E1 -12872.448,E2 -12872.448} C_VEL
LIN {X 0,Y 369.092,Z 501.055,A -85,B 0,C 180,E1 -12874.093,E2 -12874.093} C_VEL
LIN {X 0,Y 368.502,Z 508.033,A -85,B 0,C 180,E1 -12875.745,E2 -12875.745} C_VEL
LIN {X 0,Y 368.251,Z 512.598,A -85,B 0,C 180,E1 -12877.065,E2 -12877.065} C_VEL
LIN {X 0,Y 367.82,Z 517.381,A -85,B 0,C 180,E1 -12878.791,E2 -12878.791} C_VEL
LIN {X 0,Y 367.643,Z 519.799,A -85,B 0,C 180,E1 -12879.905,E2 -12879.905} C_VEL
LIN {X 0,Y 367.498,Z 521.783,A -85,B 0,C 180,E1 -12881.023,E2 -12881.023} C_VEL
LIN {X 0,Y 367.395,Z 523.9,A -85,B 0,C 180,E1 -12882.686,E2 -12882.686} C_VEL
LIN {X 0,Y 367.279,Z 525.112,A -85,B 0,C 180,E1 -12884.402,E2 -12884.402} C_VEL
LIN {X 0,Y 367.304,Z 525.396,A -85,B 0,C 180,E1 -12885.536,E2 -12885.536} C_VEL
LIN {X 0,Y 367.344,Z 525.13,A -85,B 0,C 180,E1 -12886.943,E2 -12886.943} C_VEL
